LIN {X 0,Y 536.387,Z 823.114,A -85,B 0,C 180,E1 -258.059,E2 -258.059} C_VEL
LIN {X 0,Y 536.157,Z 833.006,A -85,B 0,C 180,E1 -259.949,E2 -259.949} C_VEL
LIN {X 0,Y 536.017,Z 840.915,A -85,B 0,C 180,E1 -261.85,E2 -261.85} C_VEL
LIN {X 0,Y 535.953,Z 847.088,A -85,B 0,C 180,E1 -263.789,E2 -263.789} C_VEL
LIN {X 0,Y 535.924,Z 851.492,A -85,B 0,C 180,E1 -265.721,E2 -265.721} C_VEL
LIN {X 0,Y 535.914,Z 854.356,A -85,B 0,C 180,E1 -267.755,E2 -267.755} C_VEL
LIN {X 0,Y 535.911,Z 855.453,A -85,B 0,C 180,E1 -269.787,E2 -269.787} C_VEL
LIN {X 0,Y 535.913,Z 854.809,A -85,B 0,C 180,E1 -271.818,E2 -271.818} C_VEL
LIN {X 0,Y 535.915,Z 852.571,A -85,B 0,C 180,E1 -273.744,E2 -273.744} C_VEL
LIN {X 0,Y 535.934,Z 848.705,A -85,B 0,C 180,E1 -275.675,E2 -275.675} C_VEL
LIN {X 0,Y 535.992,Z 843.122,A -85,B 0,C 180,E1 -277.611,E2 -277.611} C_VEL
LIN {X 0,Y 536.104,Z 835.67,A -85,B 0,C 180,E1 -279.555,E2 -279.555} C_VEL
LIN {X 0,Y 536.296,Z 826.694,A -85,B 0,C 180,E1 -281.398,E2 -281.398} C_VEL
LIN {X 0,Y 536.575,Z 816.255,A -85,B 0,C 180,E1 -283.141,E2 -283.141} C_VEL
LIN {X 0,Y 536.94,Z 804.373,A -85,B 0,C 180,E1 -284.781,E2 -284.781} C_VEL
LIN {X 0,Y 537.402,Z 790.987,A -85,B 0,C 180,E1 -286.317,E2 -286.317} C_VEL
LIN {X 0,Y 537.942,Z 775.934,A -85,B 0,C 180,E1 -287.748,E2 -287.748} C_VEL
LIN {X 0,Y 538.493,Z 760.519,A -85,B 0,C 180,E1 -288.962,E2 -288.962} C_VEL
LIN {X 0,Y 539.019,Z 744.186,A -85,B 0,C 180,E1 -290.019,E2 -290.019} C_VEL
LIN {X 0,Y 539.579,Z 727.091,A -85,B 0,C 180,E1 -290.904,E2 -290.904} C_VEL
LIN {X 0,Y 540.061,Z 708.873,A -85,B 0,C 180,E1 -291.632,E2 -291.632} C_VEL
LIN {X 0,Y 540.458,Z 689.501,A -85,B 0,C 180,E1 -292.184,E2 -292.184} C_VEL
LIN {X 0,Y 540.712,Z 668.628,A -85,B 0,C 180,E1 -292.553,E2 -292.553} C_VEL
LIN {X 0,Y 541.759,Z 481.528,A -85,B 0,C 180,E1 -295.18,E2 -295.18} C_VEL
LIN {X 0,Y 540.704,Z 474.497,A -85,B 0,C 180,E1 -295.347,E2 -295.347} C_VEL
LIN {X 0,Y 541.808,Z 432.243,A -85,B 0,C 180,E1 -298.432,E2 -298.432} C_VEL
LIN {X 0,Y 542.888,Z 388.213,A -85,B 0,C 180,E1 -301.662,E2 -301.662} C_VEL
LIN {X 0,Y 542.864,Z 381.603,A -85,B 0,C 180,E1 -302.16,E2 -302.16} C_VEL
LIN {X 0,Y 536.405,Z 363.919,A -85,B 0,C 180,E1 -303.915,E2 -303.915} C_VEL
LIN {X 0,Y 536.456,Z 363.914,A -85,B 0,C 180,E1 -307.264,E2 -307.264} C_VEL
LIN {X 0,Y 536.412,Z 363.912,A -85,B 0,C 180,E1 -310.491,E2 -310.491} C_VEL
LIN {X 0,Y 536.412,Z 363.907,A -85,B 0,C 180,E1 -313.987,E2 -313.987} C_VEL
LIN {X 0,Y 536.457,Z 363.908,A -85,B 0,C 180,E1 -317.252,E2 -317.252} C_VEL
LIN {X 0,Y 536.403,Z 363.915,A -85,B 0,C 180,E1 -320.533,E2 -320.533} C_VEL
LIN {X 0,Y 536.486,Z 364.089,A -85,B 0,C 180,E1 -323.676,E2 -323.676} C_VEL
LIN {X 0,Y 544.504,Z 385.078,A -85,B 0,C 180,E1 -326.099,E2 -326.099} C_VEL
LIN {X 0,Y 543.343,Z 422.568,A -85,B 0,C 180,E1 -329.108,E2 -329.108} C_VEL
LIN {X 0,Y 541.867,Z 466.231,A -85,B 0,C 180,E1 -332.567,E2 -332.567} C_VEL
LIN {X 0,Y 540.509,Z 512.697,A -85,B 0,C 180,E1 -336.159,E2 -336.159} C_VEL
LIN {X 0,Y 539.079,Z 559.766,A -85,B 0,C 180,E1 -339.803,E2 -339.803} C_VEL
LIN {X 0,Y 538.459,Z 589.965,A -85,B 0,C 180,E1 -342.057,E2 -342.057} C_VEL
LIN {X 0,Y 539.022,Z 598.616,A -85,B 0,C 180,E1 -342.216,E2 -342.216} C_VEL
LIN {X 0,Y 538.33,Z 729.225,A -85,B 0,C 180,E1 -344.027,E2 -344.027} C_VEL
LIN {X 0,Y 538.167,Z 742.956,A -85,B 0,C 180,E1 -344.34,E2 -344.34} C_VEL
LIN {X 0,Y 537.937,Z 758.206,A -85,B 0,C 180,E1 -344.862,E2 -344.862} C_VEL
LIN {X 0,Y 537.587,Z 772.683,A -85,B 0,C 180,E1 -345.568,E2 -345.568} C_VEL
LIN {X 0,Y 537.284,Z 784.959,A -85,B 0,C 180,E1 -346.329,E2 -346.329} C_VEL
LIN {X 0,Y 536.974,Z 797.896,A -85,B 0,C 180,E1 -347.307,E2 -347.307} C_VEL
LIN {X 0,Y 536.642,Z 810.315,A -85,B 0,C 180,E1 -348.5,E2 -348.5} C_VEL
LIN {X 0,Y 536.416,Z 819.61,A -85,B 0,C 180,E1 -349.583,E2 -349.583} C_VEL
LIN {X 0,Y 536.231,Z 828.137,A -85,B 0,C 180,E1 -350.772,E2 -350.772} C_VEL
LIN {X 0,Y 536.079,Z 836.92,A -85,B 0,C 180,E1 -352.282,E2 -352.282} C_VEL
LIN {X 0,Y 535.984,Z 843.614,A -85,B 0,C 180,E1 -353.788,E2 -353.788} C_VEL
LIN {X 0,Y 535.941,Z 848.401,A -85,B 0,C 180,E1 -355.184,E2 -355.184} C_VEL
LIN {X 0,Y 535.919,Z 852.383,A -85,B 0,C 180,E1 -356.791,E2 -356.791} C_VEL
LIN {X 0,Y 535.916,Z 854.749,A -85,B 0,C 180,E1 -358.503,E2 -358.503} C_VEL
LIN {X 0,Y 535.917,Z 855.42,A -85,B 0,C 180,E1 -360,E2 -360} C_VEL
LIN {X 0,Y 535.915,Z 854.816,A -85,B 0,C 180,E1 -361.496,E2 -361.496} C_VEL
LIN {X 0,Y 535.921,Z 852.56,A -85,B 0,C 180,E1 -363.208,E2 -363.208} C_VEL
LIN {X 0,Y 535.941,Z 848.675,A -85,B 0,C 180,E1 -364.815,E2 -364.815} C_VEL
LIN {X 0,Y 535.978,Z 843.962,A -85,B 0,C 180,E1 -366.211,E2 -366.211} C_VEL
LIN {X 0,Y 536.062,Z 837.86,A -85,B 0,C 180,E1 -367.61,E2 -367.61} C_VEL
LIN {X 0,Y 536.223,Z 828.743,A -85,B 0,C 180,E1 -369.227,E2 -369.227} C_VEL
LIN {X 0,Y 536.4,Z 820.32,A -85,B 0,C 180,E1 -370.417,E2 -370.417} C_VEL
LIN {X 0,Y 536.62,Z 811.143,A -85,B 0,C 180,E1 -371.5,E2 -371.5} C_VEL
LIN {X 0,Y 536.925,Z 799.619,A -85,B 0,C 180,E1 -372.631,E2 -372.631} C_VEL
LIN {X 0,Y 537.274,Z 785.525,A -85,B 0,C 180,E1 -373.726,E2 -373.726} C_VEL
LIN {X 0,Y 537.565,Z 774.465,A -85,B 0,C 180,E1 -374.432,E2 -374.432} C_VEL
LIN {X 0,Y 537.878,Z 761.699,A -85,B 0,C 180,E1 -375.084,E2 -375.084} C_VEL
LIN {X 0,Y 538.172,Z 745.734,A -85,B 0,C 180,E1 -375.687,E2 -375.687} C_VEL
LIN {X 0,Y 538.345,Z 730.703,A -85,B 0,C 180,E1 -376.048,E2 -376.048} C_VEL
LIN {X 0,Y 539.112,Z 638.988,A -85,B 0,C 180,E1 -377.399,E2 -377.399} C_VEL
LIN {X 0,Y 539.332,Z 593.98,A -85,B 0,C 180,E1 -378.066,E2 -378.066} C_VEL
LIN {X 0,Y 539.288,Z 591.918,A -85,B 0,C 180,E1 -378.148,E2 -378.148} C_VEL
LIN {X 0,Y 541.136,Z 554.692,A -85,B 0,C 180,E1 -381.175,E2 -381.175} C_VEL
LIN {X 0,Y 544.018,Z 511.719,A -85,B 0,C 180,E1 -384.778,E2 -384.778} C_VEL
LIN {X 0,Y 547.31,Z 475.035,A -85,B 0,C 180,E1 -388.002,E2 -388.002} C_VEL
LIN {X 0,Y 551.674,Z 441.606,A -85,B 0,C 180,E1 -391.1,E2 -391.1} C_VEL
LIN {X 0,Y 556.543,Z 416.023,A -85,B 0,C 180,E1 -393.658,E2 -393.658} C_VEL
LIN {X 0,Y 558.549,Z 407.726,A -85,B 0,C 180,E1 -394.573,E2 -394.573} C_VEL
LIN {X 0,Y 559.455,Z 403.927,A -85,B 0,C 180,E1 -395.061,E2 -395.061} C_VEL
LIN {X 0,Y 558.872,Z 401.471,A -85,B 0,C 180,E1 -395.931,E2 -395.931} C_VEL
LIN {X 0,Y 558.829,Z 399.609,A -85,B 0,C 180,E1 -397.082,E2 -397.082} C_VEL
LIN {X 0,Y 559.096,Z 399.371,A -85,B 0,C 180,E1 -397.474,E2 -397.474} C_VEL
LIN {X 0,Y 554.148,Z 410.442,A -85,B 0,C 180,E1 -398.498,E2 -398.498} C_VEL
LIN {X 0,Y 550.307,Z 424.122,A -85,B 0,C 180,E1 -399.623,E2 -399.623} C_VEL
LIN {X 0,Y 547.791,Z 440.126,A -85,B 0,C 180,E1 -400.829,E2 -400.829} C_VEL
LIN {X 0,Y 547.322,Z 456.11,A -85,B 0,C 180,E1 -402.023,E2 -402.023} C_VEL
LIN {X 0,Y 548.928,Z 469.64,A -85,B 0,C 180,E1 -403.082,E2 -403.082} C_VEL
LIN {X 0,Y 552.062,Z 480.529,A -85,B 0,C 180,E1 -403.993,E2 -403.993} C_VEL
LIN {X 0,Y 556.38,Z 489.245,A -85,B 0,C 180,E1 -404.785,E2 -404.785} C_VEL
LIN {X 0,Y 562.574,Z 497.444,A -85,B 0,C 180,E1 -405.6,E2 -405.6} C_VEL
LIN {X 0,Y 569.615,Z 503.816,A -85,B 0,C 180,E1 -406.318,E2 -406.318} C_VEL
LIN {X 0,Y 577.113,Z 508.538,A -85,B 0,C 180,E1 -406.98,E2 -406.98} C_VEL
LIN {X 0,Y 581.203,Z 510.142,A -85,B 0,C 180,E1 -407.461,E2 -407.461} C_VEL
LIN {X 0,Y 584.395,Z 510.594,A -85,B 0,C 180,E1 -408.012,E2 -408.012} C_VEL
LIN {X 0,Y 586.46,Z 509.917,A -85,B 0,C 180,E1 -408.604,E2 -408.604} C_VEL
LIN {X 0,Y 587.224,Z 508.161,A -85,B 0,C 180,E1 -409.215,E2 -409.215} C_VEL
LIN {X 0,Y 586.511,Z 505.309,A -85,B 0,C 180,E1 -409.815,E2 -409.815} C_VEL
LIN {X 0,Y 584.311,Z 501.673,A -85,B 0,C 180,E1 -410.337,E2 -410.337} C_VEL
LIN {X 0,Y 578.602,Z 493.885,A -85,B 0,C 180,E1 -411.054,E2 -411.054} C_VEL
LIN {X 0,Y 573.375,Z 484.319,A -85,B 0,C 180,E1 -411.705,E2 -411.705} C_VEL
LIN {X 0,Y 569.141,Z 473.459,A -85,B 0,C 180,E1 -412.248,E2 -412.248} C_VEL
LIN {X 0,Y 565.904,Z 461.458,A -85,B 0,C 180,E1 -412.673,E2 -412.673} C_VEL
LIN {X 0,Y 564.883,Z 456.447,A -85,B 0,C 180,E1 -412.809,E2 -412.809} C_VEL
LIN {X 0,Y 562.174,Z 463.362,A -85,B 0,C 180,E1 -413.175,E2 -413.175} C_VEL
LIN {X 0,Y 559.86,Z 469.22,A -85,B 0,C 180,E1 -413.492,E2 -413.492} C_VEL
LIN {X 0,Y 558.97,Z 470.969,A -85,B 0,C 180,E1 -413.615,E2 -413.615} C_VEL
LIN {X 0,Y 554.81,Z 519.429,A -85,B 0,C 180,E1 -414.203,E2 -414.203} C_VEL
LIN {X 0,Y 551.082,Z 552.372,A -85,B 0,C 180,E1 -414.744,E2 -414.744} C_VEL
LIN {X 0,Y 548.664,Z 567.257,A -85,B 0,C 180,E1 -415.102,E2 -415.102} C_VEL
LIN {X 0,Y 547.486,Z 570.982,A -85,B 0,C 180,E1 -415.279,E2 -415.279} C_VEL
LIN {X 0,Y 547.134,Z 571.563,A -85,B 0,C 180,E1 -415.337,E2 -415.337} C_VEL
LIN {X 0,Y 545.349,Z 761.519,A -85,B 0,C 180,E1 -418.174,E2 -418.174} C_VEL
LIN {X 0,Y 544.771,Z 783.502,A -85,B 0,C 180,E1 -418.695,E2 -418.695} C_VEL
LIN {X 0,Y 544.053,Z 806.31,A -85,B 0,C 180,E1 -419.459,E2 -419.459} C_VEL
LIN {X 0,Y 543.205,Z 827.548,A -85,B 0,C 180,E1 -420.381,E2 -420.381} C_VEL
LIN {X 0,Y 542.286,Z 847.779,A -85,B 0,C 180,E1 -421.475,E2 -421.475} C_VEL
LIN {X 0,Y 541.287,Z 867.98,A -85,B 0,C 180,E1 -422.794,E2 -422.794} C_VEL
LIN {X 0,Y 540.249,Z 887.816,A -85,B 0,C 180,E1 -424.337,E2 -424.337} C_VEL
LIN {X 0,Y 539.331,Z 905.831,A -85,B 0,C 180,E1 -425.988,E2 -425.988} C_VEL
LIN {X 0,Y 538.461,Z 923.22,A -85,B 0,C 180,E1 -427.855,E2 -427.855} C_VEL
LIN {X 0,Y 537.693,Z 939.401,A -85,B 0,C 180,E1 -429.894,E2 -429.894} C_VEL
LIN {X 0,Y 537.082,Z 953.596,A -85,B 0,C 180,E1 -431.999,E2 -431.999} C_VEL
LIN {X 0,Y 536.623,Z 966.268,A -85,B 0,C 180,E1 -434.214,E2 -434.214} C_VEL
LIN {X 0,Y 536.313,Z 976.854,A -85,B 0,C 180,E1 -436.414,E2 -436.414} C_VEL
LIN {X 0,Y 536.107,Z 985.923,A -85,B 0,C 180,E1 -438.707,E2 -438.707} C_VEL
LIN {X 0,Y 535.994,Z 993.093,A -85,B 0,C 180,E1 -440.985,E2 -440.985} C_VEL
LIN {X 0,Y 535.942,Z 998.591,A -85,B 0,C 180,E1 -443.25,E2 -443.25} C_VEL
LIN {X 0,Y 535.921,Z 1002.584,A -85,B 0,C 180,E1 -445.613,E2 -445.613} C_VEL
LIN {X 0,Y 535.911,Z 1004.832,A -85,B 0,C 180,E1 -447.968,E2 -447.968} C_VEL
LIN {X 0,Y 535.894,Z 1005.442,A -85,B 0,C 180,E1 -450.427,E2 -450.427} C_VEL
LIN {X 0,Y 535.894,Z 1004.424,A -85,B 0,C 180,E1 -452.673,E2 -452.673} C_VEL
LIN {X 0,Y 535.901,Z 1001.8,A -85,B 0,C 180,E1 -454.926,E2 -454.926} C_VEL
LIN {X 0,Y 535.929,Z 997.683,A -85,B 0,C 180,E1 -457.18,E2 -457.18} C_VEL
LIN {X 0,Y 535.997,Z 991.879,A -85,B 0,C 180,E1 -459.448,E2 -459.448} C_VEL
LIN {X 0,Y 536.128,Z 984.297,A -85,B 0,C 180,E1 -461.735,E2 -461.735} C_VEL
LIN {X 0,Y 536.357,Z 974.911,A -85,B 0,C 180,E1 -464.025,E2 -464.025} C_VEL
LIN {X 0,Y 536.693,Z 963.937,A -85,B 0,C 180,E1 -466.227,E2 -466.227} C_VEL
LIN {X 0,Y 537.16,Z 951.48,A -85,B 0,C 180,E1 -468.335,E2 -468.335} C_VEL
LIN {X 0,Y 537.766,Z 937.595,A -85,B 0,C 180,E1 -470.346,E2 -470.346} C_VEL
LIN {X 0,Y 538.505,Z 922.234,A -85,B 0,C 180,E1 -472.257,E2 -472.257} C_VEL
LIN {X 0,Y 539.363,Z 905.276,A -85,B 0,C 180,E1 -474.068,E2 -474.068} C_VEL
LIN {X 0,Y 540.321,Z 886.47,A -85,B 0,C 180,E1 -475.776,E2 -475.776} C_VEL
LIN {X 0,Y 541.326,Z 867.187,A -85,B 0,C 180,E1 -477.262,E2 -477.262} C_VEL
LIN {X 0,Y 542.328,Z 846.795,A -85,B 0,C 180,E1 -478.582,E2 -478.582} C_VEL
LIN {X 0,Y 543.204,Z 827.56,A -85,B 0,C 180,E1 -479.618,E2 -479.618} C_VEL
LIN {X 0,Y 544.053,Z 806.327,A -85,B 0,C 180,E1 -480.54,E2 -480.54} C_VEL
LIN {X 0,Y 544.782,Z 783.156,A -85,B 0,C 180,E1 -481.315,E2 -481.315} C_VEL
LIN {X 0,Y 545.362,Z 761.024,A -85,B 0,C 180,E1 -481.836,E2 -481.836} C_VEL
LIN {X 0,Y 547.27,Z 571.184,A -85,B 0,C 180,E1 -484.688,E2 -484.688} C_VEL
LIN {X 0,Y 548.267,Z 568.899,A -85,B 0,C 180,E1 -484.838,E2 -484.838} C_VEL
LIN {X 0,Y 550.436,Z 557.003,A -85,B 0,C 180,E1 -485.161,E2 -485.161} C_VEL
LIN {X 0,Y 553.985,Z 527.566,A -85,B 0,C 180,E1 -485.679,E2 -485.679} C_VEL
LIN {X 0,Y 558.161,Z 481.457,A -85,B 0,C 180,E1 -486.272,E2 -486.272} C_VEL
LIN {X 0,Y 559.115,Z 470.446,A -85,B 0,C 180,E1 -486.405,E2 -486.405} C_VEL
LIN {X 0,Y 561.46,Z 465.551,A -85,B 0,C 180,E1 -486.728,E2 -486.728} C_VEL
LIN {X 0,Y 563.371,Z 460.11,A -85,B 0,C 180,E1 -486.988,E2 -486.988} C_VEL
LIN {X 0,Y 564.936,Z 456.583,A -85,B 0,C 180,E1 -487.198,E2 -487.198} C_VEL
LIN {X 0,Y 567.839,Z 469.202,A -85,B 0,C 180,E1 -487.582,E2 -487.582} C_VEL
LIN {X 0,Y 571.748,Z 480.579,A -85,B 0,C 180,E1 -488.088,E2 -488.088} C_VEL
LIN {X 0,Y 576.639,Z 490.657,A -85,B 0,C 180,E1 -488.704,E2 -488.704} C_VEL
LIN {X 0,Y 582.546,Z 499.398,A -85,B 0,C 180,E1 -489.424,E2 -489.424} C_VEL
LIN {X 0,Y 585.465,Z 503.391,A -85,B 0,C 180,E1 -489.884,E2 -489.884} C_VEL
LIN {X 0,Y 586.997,Z 506.612,A -85,B 0,C 180,E1 -490.429,E2 -490.429} C_VEL
LIN {X 0,Y 587.094,Z 508.969,A -85,B 0,C 180,E1 -491.022,E2 -491.022} C_VEL
LIN {X 0,Y 585.831,Z 510.295,A -85,B 0,C 180,E1 -491.622,E2 -491.622} C_VEL
LIN {X 0,Y 583.164,Z 510.544,A -85,B 0,C 180,E1 -492.229,E2 -492.229} C_VEL
LIN {X 0,Y 579.798,Z 509.694,A -85,B 0,C 180,E1 -492.724,E2 -492.724} C_VEL
LIN {X 0,Y 571.887,Z 505.541,A -85,B 0,C 180,E1 -493.63,E2 -493.63} C_VEL
LIN {X 0,Y 565.274,Z 499.908,A -85,B 0,C 180,E1 -494.535,E2 -494.535} C_VEL
LIN {X 0,Y 560.009,Z 492.953,A -85,B 0,C 180,E1 -495.439,E2 -495.439} C_VEL
LIN {X 0,Y 555.868,Z 484.228,A -85,B 0,C 180,E1 -496.385,E2 -496.385} C_VEL
LIN {X 0,Y 553.159,Z 473.762,A -85,B 0,C 180,E1 -497.363,E2 -497.363} C_VEL
LIN {X 0,Y 551.719,Z 460.276,A -85,B 0,C 180,E1 -498.457,E2 -498.457} C_VEL
LIN {X 0,Y 551.957,Z 441.599,A -85,B 0,C 180,E1 -499.775,E2 -499.775} C_VEL
LIN {X 0,Y 553.891,Z 401.672,A -85,B 0,C 180,E1 -502.531,E2 -502.531} C_VEL
LIN {X 0,Y 554.042,Z 396.212,A -85,B 0,C 180,E1 -502.933,E2 -502.933} C_VEL
LIN {X 0,Y 546.158,Z 382.054,A -85,B 0,C 180,E1 -505.04,E2 -505.04} C_VEL
LIN {X 0,Y 541.163,Z 373.11,A -85,B 0,C 180,E1 -506.436,E2 -506.436} C_VEL
LIN {X 0,Y 539.331,Z 369.712,A -85,B 0,C 180,E1 -506.973,E2 -506.973} C_VEL
LIN {X 0,Y 536.8,Z 365.411,A -85,B 0,C 180,E1 -507.685,E2 -507.685} C_VEL
LIN {X 0,Y 536.468,Z 363.913,A -85,B 0,C 180,E1 -507.87,E2 -507.87} C_VEL
LIN {X 0,Y 536.425,Z 363.915,A -85,B 0,C 180,E1 -511.257,E2 -511.257} C_VEL
LIN {X 0,Y 536.433,Z 363.914,A -85,B 0,C 180,E1 -514.852,E2 -514.852} C_VEL
LIN {X 0,Y 536.465,Z 363.91,A -85,B 0,C 180,E1 -518.23,E2 -518.23} C_VEL
LIN {X 0,Y 536.442,Z 363.914,A -85,B 0,C 180,E1 -521.752,E2 -521.752} C_VEL
LIN {X 0,Y 536.466,Z 363.912,A -85,B 0,C 180,E1 -525.096,E2 -525.096} C_VEL
LIN {X 0,Y 536.46,Z 363.913,A -85,B 0,C 180,E1 -528.497,E2 -528.497} C_VEL
LIN {X 0,Y 536.458,Z 363.913,A -85,B 0,C 180,E1 -531.857,E2 -531.857} C_VEL
LIN {X 0,Y 536.44,Z 363.917,A -85,B 0,C 180,E1 -535.189,E2 -535.189} C_VEL
LIN {X 0,Y 536.461,Z 363.914,A -85,B 0,C 180,E1 -538.505,E2 -538.505} C_VEL
LIN {X 0,Y 536.422,Z 363.918,A -85,B 0,C 180,E1 -541.923,E2 -541.923} C_VEL
LIN {X 0,Y 536.455,Z 363.911,A -85,B 0,C 180,E1 -545.348,E2 -545.348} C_VEL
LIN {X 0,Y 536.43,Z 363.915,A -85,B 0,C 180,E1 -548.684,E2 -548.684} C_VEL
LIN {X 0,Y 536.427,Z 363.915,A -85,B 0,C 180,E1 -552.159,E2 -552.159} C_VEL
LIN {X 0,Y 536.466,Z 363.909,A -85,B 0,C 180,E1 -555.569,E2 -555.569} C_VEL
LIN {X 0,Y 536.438,Z 363.914,A -85,B 0,C 180,E1 -559.037,E2 -559.037} C_VEL
LIN {X 0,Y 536.465,Z 363.914,A -85,B 0,C 180,E1 -562.463,E2 -562.463} C_VEL
LIN {X 0,Y 536.459,Z 363.913,A -85,B 0,C 180,E1 -565.858,E2 -565.858} C_VEL
LIN {X 0,Y 536.457,Z 363.913,A -85,B 0,C 180,E1 -569.277,E2 -569.277} C_VEL
LIN {X 0,Y 536.432,Z 363.916,A -85,B 0,C 180,E1 -572.597,E2 -572.597} C_VEL
LIN {X 0,Y 536.433,Z 363.91,A -85,B 0,C 180,E1 -574.588,E2 -574.588} C_VEL
LIN {X 0,Y 535.428,Z 364.033,A -85,B 0,C 180,E1 -575.411,E2 -575.411} C_VEL
LIN {X 0,Y 529.04,Z 364.829,A -85,B 0,C 180,E1 -577.723,E2 -577.723} C_VEL
LIN {X 0,Y 528.526,Z 364.894,A -85,B 0,C 180,E1 -578.325,E2 -578.325} C_VEL
LIN {X 0,Y 528.504,Z 364.893,A -85,B 0,C 180,E1 -581.807,E2 -581.807} C_VEL
LIN {X 0,Y 528.523,Z 364.905,A -85,B 0,C 180,E1 -585.188,E2 -585.188} C_VEL
LIN {X 0,Y 528.521,Z 364.904,A -85,B 0,C 180,E1 -588.682,E2 -588.682} C_VEL
LIN {X 0,Y 528.513,Z 364.899,A -85,B 0,C 180,E1 -592.083,E2 -592.083} C_VEL
LIN {X 0,Y 528.479,Z 364.909,A -85,B 0,C 180,E1 -595.55,E2 -595.55} C_VEL
LIN {X 0,Y 528.496,Z 365.068,A -85,B 0,C 180,E1 -595.715,E2 -595.715} C_VEL
LIN {X 0,Y 535.912,Z 384.982,A -85,B 0,C 180,E1 -597.708,E2 -597.708} C_VEL
LIN {X 0,Y 534.68,Z 430.458,A -85,B 0,C 180,E1 -601.087,E2 -601.087} C_VEL
LIN {X 0,Y 533.602,Z 476.361,A -85,B 0,C 180,E1 -604.403,E2 -604.403} C_VEL
LIN {X 0,Y 534.725,Z 485.378,A -85,B 0,C 180,E1 -604.596,E2 -604.596} C_VEL
LIN {X 0,Y 533.229,Z 683.64,A -85,B 0,C 180,E1 -607.434,E2 -607.434} C_VEL
LIN {X 0,Y 532.889,Z 701.992,A -85,B 0,C 180,E1 -607.885,E2 -607.885} C_VEL
LIN {X 0,Y 532.411,Z 719.706,A -85,B 0,C 180,E1 -608.518,E2 -608.518} C_VEL
LIN {X 0,Y 531.792,Z 737.309,A -85,B 0,C 180,E1 -609.358,E2 -609.358} C_VEL
LIN {X 0,Y 531.116,Z 753.841,A -85,B 0,C 180,E1 -610.365,E2 -610.365} C_VEL
LIN {X 0,Y 530.393,Z 771.626,A -85,B 0,C 180,E1 -611.707,E2 -611.707} C_VEL
LIN {X 0,Y 529.791,Z 786.298,A -85,B 0,C 180,E1 -613.048,E2 -613.048} C_VEL
LIN {X 0,Y 529.247,Z 800.016,A -85,B 0,C 180,E1 -614.551,E2 -614.551} C_VEL
LIN {X 0,Y 528.786,Z 812.65,A -85,B 0,C 180,E1 -616.217,E2 -616.217} C_VEL
LIN {X 0,Y 528.433,Z 823.943,A -85,B 0,C 180,E1 -618.023,E2 -618.023} C_VEL
LIN {X 0,Y 528.187,Z 833.309,A -85,B 0,C 180,E1 -619.861,E2 -619.861} C_VEL
LIN {X 0,Y 528.038,Z 840.916,A -85,B 0,C 180,E1 -621.726,E2 -621.726} C_VEL
LIN {X 0,Y 527.958,Z 847.09,A -85,B 0,C 180,E1 -623.694,E2 -623.694} C_VEL
LIN {X 0,Y 527.925,Z 851.494,A -85,B 0,C 180,E1 -625.656,E2 -625.656} C_VEL
LIN {X 0,Y 527.913,Z 854.356,A -85,B 0,C 180,E1 -627.721,E2 -627.721} C_VEL
LIN {X 0,Y 527.911,Z 855.453,A -85,B 0,C 180,E1 -629.783,E2 -629.783} C_VEL
LIN {X 0,Y 527.913,Z 854.808,A -85,B 0,C 180,E1 -631.845,E2 -631.845} C_VEL
LIN {X 0,Y 527.918,Z 852.57,A -85,B 0,C 180,E1 -633.801,E2 -633.801} C_VEL
LIN {X 0,Y 527.937,Z 848.704,A -85,B 0,C 180,E1 -635.761,E2 -635.761} C_VEL
LIN {X 0,Y 528.007,Z 843.119,A -85,B 0,C 180,E1 -637.727,E2 -637.727} C_VEL
LIN {X 0,Y 528.134,Z 835.669,A -85,B 0,C 180,E1 -639.701,E2 -639.701} C_VEL
LIN {X 0,Y 528.354,Z 826.693,A -85,B 0,C 180,E1 -641.572,E2 -641.572} C_VEL
LIN {X 0,Y 528.674,Z 816.253,A -85,B 0,C 180,E1 -643.341,E2 -643.341} C_VEL
LIN {X 0,Y 529.111,Z 803.908,A -85,B 0,C 180,E1 -645.063,E2 -645.063} C_VEL
LIN {X 0,Y 529.633,Z 790.432,A -85,B 0,C 180,E1 -646.619,E2 -646.619} C_VEL
LIN {X 0,Y 530.222,Z 775.924,A -85,B 0,C 180,E1 -648.015,E2 -648.015} C_VEL
LIN {X 0,Y 530.88,Z 759.69,A -85,B 0,C 180,E1 -649.307,E2 -649.307} C_VEL
LIN {X 0,Y 531.528,Z 743.735,A -85,B 0,C 180,E1 -650.366,E2 -650.366} C_VEL
LIN {X 0,Y 532.184,Z 726.55,A -85,B 0,C 180,E1 -651.27,E2 -651.27} C_VEL
LIN {X 0,Y 532.732,Z 708.036,A -85,B 0,C 180,E1 -652.011,E2 -652.011} C_VEL
LIN {X 0,Y 533.133,Z 689.61,A -85,B 0,C 180,E1 -652.531,E2 -652.531} C_VEL
LIN {X 0,Y 533.377,Z 668.55,A -85,B 0,C 180,E1 -652.897,E2 -652.897} C_VEL
LIN {X 0,Y 534.562,Z 482.581,A -85,B 0,C 180,E1 -655.544,E2 -655.544} C_VEL
LIN {X 0,Y 533.518,Z 475.565,A -85,B 0,C 180,E1 -655.719,E2 -655.719} C_VEL
LIN {X 0,Y 534.694,Z 430.123,A -85,B 0,C 180,E1 -659.03,E2 -659.03} C_VEL
LIN {X 0,Y 535.897,Z 385.079,A -85,B 0,C 180,E1 -662.377,E2 -662.377} C_VEL
LIN {X 0,Y 529.73,Z 368.431,A -85,B 0,C 180,E1 -664.044,E2 -664.044} C_VEL
LIN {X 0,Y 528.481,Z 364.904,A -85,B 0,C 180,E1 -664.405,E2 -664.405} C_VEL
LIN {X 0,Y 528.473,Z 364.904,A -85,B 0,C 180,E1 -667.807,E2 -667.807} C_VEL
LIN {X 0,Y 528.521,Z 364.895,A -85,B 0,C 180,E1 -671.031,E2 -671.031} C_VEL
LIN {X 0,Y 528.466,Z 364.896,A -85,B 0,C 180,E1 -674.342,E2 -674.342} C_VEL
LIN {X 0,Y 528.509,Z 364.892,A -85,B 0,C 180,E1 -677.707,E2 -677.707} C_VEL
LIN {X 0,Y 528.479,Z 364.898,A -85,B 0,C 180,E1 -680.948,E2 -680.948} C_VEL
LIN {X 0,Y 528.518,Z 365.148,A -85,B 0,C 180,E1 -683.093,E2 -683.093} C_VEL
LIN {X 0,Y 537.22,Z 387.368,A -85,B 0,C 180,E1 -685.727,E2 -685.727} C_VEL
LIN {X 0,Y 537.491,Z 389.74,A -85,B 0,C 180,E1 -685.949,E2 -685.949} C_VEL
LIN {X 0,Y 536.131,Z 429.265,A -85,B 0,C 180,E1 -689.145,E2 -689.145} C_VEL
LIN {X 0,Y 534.525,Z 472.595,A -85,B 0,C 180,E1 -692.602,E2 -692.602} C_VEL
LIN {X 0,Y 533.057,Z 517.272,A -85,B 0,C 180,E1 -696.099,E2 -696.099} C_VEL
LIN {X 0,Y 531.6,Z 563.498,A -85,B 0,C 180,E1 -699.695,E2 -699.695} C_VEL
LIN {X 0,Y 530.993,Z 590.742,A -85,B 0,C 180,E1 -701.746,E2 -701.746} C_VEL
LIN {X 0,Y 531.581,Z 599.108,A -85,B 0,C 180,E1 -701.905,E2 -701.905} C_VEL
LIN {X 0,Y 530.718,Z 728.012,A -85,B 0,C 180,E1 -703.744,E2 -703.744} C_VEL
LIN {X 0,Y 530.542,Z 742.648,A -85,B 0,C 180,E1 -704.067,E2 -704.067} C_VEL
LIN {X 0,Y 530.302,Z 757.908,A -85,B 0,C 180,E1 -704.582,E2 -704.582} C_VEL
LIN {X 0,Y 529.94,Z 772.805,A -85,B 0,C 180,E1 -705.299,E2 -705.299} C_VEL
LIN {X 0,Y 529.602,Z 785.194,A -85,B 0,C 180,E1 -706.071,E2 -706.071} C_VEL
LIN {X 0,Y 529.238,Z 797.381,A -85,B 0,C 180,E1 -707.007,E2 -707.007} C_VEL
LIN {X 0,Y 528.844,Z 809.94,A -85,B 0,C 180,E1 -708.218,E2 -708.218} C_VEL
LIN {X 0,Y 528.525,Z 819.988,A -85,B 0,C 180,E1 -709.426,E2 -709.426} C_VEL
LIN {X 0,Y 528.291,Z 828.291,A -85,B 0,C 180,E1 -710.632,E2 -710.632} C_VEL
LIN {X 0,Y 528.092,Z 837.428,A -85,B 0,C 180,E1 -712.274,E2 -712.274} C_VEL
LIN {X 0,Y 527.994,Z 843.608,A -85,B 0,C 180,E1 -713.694,E2 -713.694} C_VEL
LIN {X 0,Y 527.946,Z 848.394,A -85,B 0,C 180,E1 -715.111,E2 -715.111} C_VEL
LIN {X 0,Y 527.92,Z 852.379,A -85,B 0,C 180,E1 -716.742,E2 -716.742} C_VEL
LIN {X 0,Y 527.915,Z 854.742,A -85,B 0,C 180,E1 -718.48,E2 -718.48} C_VEL
LIN {X 0,Y 527.917,Z 855.411,A -85,B 0,C 180,E1 -720,E2 -720} C_VEL
LIN {X 0,Y 527.915,Z 854.807,A -85,B 0,C 180,E1 -721.519,E2 -721.519} C_VEL
LIN {X 0,Y 527.922,Z 852.561,A -85,B 0,C 180,E1 -723.257,E2 -723.257} C_VEL
LIN {X 0,Y 527.944,Z 848.664,A -85,B 0,C 180,E1 -724.889,E2 -724.889} C_VEL
LIN {X 0,Y 527.988,Z 843.951,A -85,B 0,C 180,E1 -726.306,E2 -726.306} C_VEL
LIN {X 0,Y 528.084,Z 837.849,A -85,B 0,C 180,E1 -727.725,E2 -727.725} C_VEL
LIN {X 0,Y 528.293,Z 829.028,A -85,B 0,C 180,E1 -729.367,E2 -729.367} C_VEL
LIN {X 0,Y 528.535,Z 820.937,A -85,B 0,C 180,E1 -730.573,E2 -730.573} C_VEL
LIN {X 0,Y 528.83,Z 812.08,A -85,B 0,C 180,E1 -731.671,E2 -731.671} C_VEL
LIN {X 0,Y 529.23,Z 800.857,A -85,B 0,C 180,E1 -732.826,E2 -732.826} C_VEL
LIN {X 0,Y 529.666,Z 787.274,A -85,B 0,C 180,E1 -733.927,E2 -733.927} C_VEL
LIN {X 0,Y 530.03,Z 774.346,A -85,B 0,C 180,E1 -734.754,E2 -734.754} C_VEL
LIN {X 0,Y 530.393,Z 759.935,A -85,B 0,C 180,E1 -735.47,E2 -735.47} C_VEL
LIN {X 0,Y 530.63,Z 744.334,A -85,B 0,C 180,E1 -736.014,E2 -736.014} C_VEL
LIN {X 0,Y 530.795,Z 729.651,A -85,B 0,C 180,E1 -736.349,E2 -736.349} C_VEL
LIN {X 0,Y 531.93,Z 628.266,A -85,B 0,C 180,E1 -737.912,E2 -737.912} C_VEL
LIN {X 0,Y 532.287,Z 594.804,A -85,B 0,C 180,E1 -738.467,E2 -738.467} C_VEL
LIN {X 0,Y 534.096,Z 563.14,A -85,B 0,C 180,E1 -741.065,E2 -741.065} C_VEL
LIN {X 0,Y 536.74,Z 524.756,A -85,B 0,C 180,E1 -744.311,E2 -744.311} C_VEL
LIN {X 0,Y 540.608,Z 484.193,A -85,B 0,C 180,E1 -747.899,E2 -747.899} C_VEL
LIN {X 0,Y 544.696,Z 453.781,A -85,B 0,C 180,E1 -750.745,E2 -750.745} C_VEL
LIN {X 0,Y 549.942,Z 426.989,A -85,B 0,C 180,E1 -753.428,E2 -753.428} C_VEL
LIN {X 0,Y 553.677,Z 413.284,A -85,B 0,C 180,E1 -754.929,E2 -754.929} C_VEL
LIN {X 0,Y 554.683,Z 409.657,A -85,B 0,C 180,E1 -755.435,E2 -755.435} C_VEL
LIN {X 0,Y 554.418,Z 407.915,A -85,B 0,C 180,E1 -756.137,E2 -756.137} C_VEL
LIN {X 0,Y 554.593,Z 406.501,A -85,B 0,C 180,E1 -757.125,E2 -757.125} C_VEL
LIN {X 0,Y 548.964,Z 417.696,A -85,B 0,C 180,E1 -758.194,E2 -758.194} C_VEL
LIN {X 0,Y 544.511,Z 431.403,A -85,B 0,C 180,E1 -759.37,E2 -759.37} C_VEL
LIN {X 0,Y 541.796,Z 446.57,A -85,B 0,C 180,E1 -760.588,E2 -760.588} C_VEL
LIN {X 0,Y 541.209,Z 461.137,A -85,B 0,C 180,E1 -761.752,E2 -761.752} C_VEL
LIN {X 0,Y 542.67,Z 474.175,A -85,B 0,C 180,E1 -762.835,E2 -762.835} C_VEL
LIN {X 0,Y 545.848,Z 485.335,A -85,B 0,C 180,E1 -763.82,E2 -763.82} C_VEL
LIN {X 0,Y 550.314,Z 494.368,A -85,B 0,C 180,E1 -764.679,E2 -764.679} C_VEL
LIN {X 0,Y 556.383,Z 502.505,A -85,B 0,C 180,E1 -765.515,E2 -765.515} C_VEL
LIN {X 0,Y 564.055,Z 509.609,A -85,B 0,C 180,E1 -766.321,E2 -766.321} C_VEL
LIN {X 0,Y 573.177,Z 515.397,A -85,B 0,C 180,E1 -767.109,E2 -767.109} C_VEL
LIN {X 0,Y 577.397,Z 517.151,A -85,B 0,C 180,E1 -767.535,E2 -767.535} C_VEL
LIN {X 0,Y 580.887,Z 517.889,A -85,B 0,C 180,E1 -768.037,E2 -768.037} C_VEL
LIN {X 0,Y 583.542,Z 517.554,A -85,B 0,C 180,E1 -768.632,E2 -768.632} C_VEL
LIN {X 0,Y 584.877,Z 516.087,A -85,B 0,C 180,E1 -769.265,E2 -769.265} C_VEL
LIN {X 0,Y 584.68,Z 513.551,A -85,B 0,C 180,E1 -769.888,E2 -769.888} C_VEL
LIN {X 0,Y 582.927,Z 510.187,A -85,B 0,C 180,E1 -770.447,E2 -770.447} C_VEL
LIN {X 0,Y 579.389,Z 505.648,A -85,B 0,C 180,E1 -770.958,E2 -770.958} C_VEL
LIN {X 0,Y 573.143,Z 496.366,A -85,B 0,C 180,E1 -771.734,E2 -771.734} C_VEL
LIN {X 0,Y 568.071,Z 485.991,A -85,B 0,C 180,E1 -772.387,E2 -772.387} C_VEL
LIN {X 0,Y 563.939,Z 474.303,A -85,B 0,C 180,E1 -772.936,E2 -772.936} C_VEL
LIN {X 0,Y 563.751,Z 473.943,A -85,B 0,C 180,E1 -772.961,E2 -772.961} C_VEL
LIN {X 0,Y 563.347,Z 476.736,A -85,B 0,C 180,E1 -773.016,E2 -773.016} C_VEL
LIN {X 0,Y 559.081,Z 524.504,A -85,B 0,C 180,E1 -773.6,E2 -773.6} C_VEL
LIN {X 0,Y 555.341,Z 556.183,A -85,B 0,C 180,E1 -774.127,E2 -774.127} C_VEL
LIN {X 0,Y 552.879,Z 570.521,A -85,B 0,C 180,E1 -774.481,E2 -774.481} C_VEL
LIN {X 0,Y 551.421,Z 575.968,A -85,B 0,C 180,E1 -774.694,E2 -774.694} C_VEL
LIN {X 0,Y 547.205,Z 626.873,A -85,B 0,C 180,E1 -775.316,E2 -775.316} C_VEL
LIN {X 0,Y 544.154,Z 647.157,A -85,B 0,C 180,E1 -775.648,E2 -775.648} C_VEL
LIN {X 0,Y 541.182,Z 660.811,A -85,B 0,C 180,E1 -776.013,E2 -776.013} C_VEL
LIN {X 0,Y 539.577,Z 667.203,A -85,B 0,C 180,E1 -776.293,E2 -776.293} C_VEL
LIN {X 0,Y 538.542,Z 761.682,A -85,B 0,C 180,E1 -777.727,E2 -777.727} C_VEL
LIN {X 0,Y 537.908,Z 783.496,A -85,B 0,C 180,E1 -778.25,E2 -778.25} C_VEL
LIN {X 0,Y 537.108,Z 806.304,A -85,B 0,C 180,E1 -779.021,E2 -779.021} C_VEL
LIN {X 0,Y 536.16,Z 827.421,A -85,B 0,C 180,E1 -779.946,E2 -779.946} C_VEL
LIN {X 0,Y 535.133,Z 847.786,A -85,B 0,C 180,E1 -781.058,E2 -781.058} C_VEL
LIN {X 0,Y 534.006,Z 867.985,A -85,B 0,C 180,E1 -782.392,E2 -782.392} C_VEL
LIN {X 0,Y 532.849,Z 887.814,A -85,B 0,C 180,E1 -783.954,E2 -783.954} C_VEL
LIN {X 0,Y 531.812,Z 905.833,A -85,B 0,C 180,E1 -785.626,E2 -785.626} C_VEL
LIN {X 0,Y 530.82,Z 923.22,A -85,B 0,C 180,E1 -787.519,E2 -787.519} C_VEL
LIN {X 0,Y 529.956,Z 939.281,A -85,B 0,C 180,E1 -789.571,E2 -789.571} C_VEL
LIN {X 0,Y 529.254,Z 953.599,A -85,B 0,C 180,E1 -791.723,E2 -791.723} C_VEL
LIN {X 0,Y 528.723,Z 966.272,A -85,B 0,C 180,E1 -793.972,E2 -793.972} C_VEL
LIN {X 0,Y 528.37,Z 976.857,A -85,B 0,C 180,E1 -796.205,E2 -796.205} C_VEL
LIN {X 0,Y 528.136,Z 985.922,A -85,B 0,C 180,E1 -798.534,E2 -798.534} C_VEL
LIN {X 0,Y 528.006,Z 993.096,A -85,B 0,C 180,E1 -800.847,E2 -800.847} C_VEL
LIN {X 0,Y 527.942,Z 998.592,A -85,B 0,C 180,E1 -803.147,E2 -803.147} C_VEL
LIN {X 0,Y 527.919,Z 1002.585,A -85,B 0,C 180,E1 -805.546,E2 -805.546} C_VEL
LIN {X 0,Y 527.912,Z 1004.834,A -85,B 0,C 180,E1 -807.937,E2 -807.937} C_VEL
LIN {X 0,Y 527.894,Z 1005.445,A -85,B 0,C 180,E1 -810.434,E2 -810.434} C_VEL
LIN {X 0,Y 527.894,Z 1004.33,A -85,B 0,C 180,E1 -812.822,E2 -812.822} C_VEL
LIN {X 0,Y 527.9,Z 1001.648,A -85,B 0,C 180,E1 -815.107,E2 -815.107} C_VEL
LIN {X 0,Y 527.938,Z 997.194,A -85,B 0,C 180,E1 -817.509,E2 -817.509} C_VEL
LIN {X 0,Y 528.021,Z 991.252,A -85,B 0,C 180,E1 -819.812,E2 -819.812} C_VEL
LIN {X 0,Y 528.185,Z 983.509,A -85,B 0,C 180,E1 -822.129,E2 -822.129} C_VEL
LIN {X 0,Y 528.466,Z 973.876,A -85,B 0,C 180,E1 -824.462,E2 -824.462} C_VEL
LIN {X 0,Y 528.878,Z 962.746,A -85,B 0,C 180,E1 -826.7,E2 -826.7} C_VEL
LIN {X 0,Y 529.457,Z 949.347,A -85,B 0,C 180,E1 -828.954,E2 -828.954} C_VEL
LIN {X 0,Y 530.165,Z 934.977,A -85,B 0,C 180,E1 -831.007,E2 -831.007} C_VEL
LIN {X 0,Y 531.038,Z 918.949,A -85,B 0,C 180,E1 -832.971,E2 -832.971} C_VEL
LIN {X 0,Y 532.065,Z 901.316,A -85,B 0,C 180,E1 -834.818,E2 -834.818} C_VEL
LIN {X 0,Y 533.153,Z 883.048,A -85,B 0,C 180,E1 -836.449,E2 -836.449} C_VEL
LIN {X 0,Y 534.243,Z 863.938,A -85,B 0,C 180,E1 -837.897,E2 -837.897} C_VEL
LIN {X 0,Y 535.321,Z 843.801,A -85,B 0,C 180,E1 -839.175,E2 -839.175} C_VEL
LIN {X 0,Y 536.394,Z 822.663,A -85,B 0,C 180,E1 -840.279,E2 -840.279} C_VEL
LIN {X 0,Y 537.288,Z 801.75,A -85,B 0,C 180,E1 -841.154,E2 -841.154} C_VEL
LIN {X 0,Y 538.052,Z 779.811,A -85,B 0,C 180,E1 -841.854,E2 -841.854} C_VEL
LIN {X 0,Y 538.609,Z 757.854,A -85,B 0,C 180,E1 -842.344,E2 -842.344} C_VEL
LIN {X 0,Y 539.718,Z 666.089,A -85,B 0,C 180,E1 -843.744,E2 -843.744} C_VEL
LIN {X 0,Y 541.823,Z 658.169,A -85,B 0,C 180,E1 -844.076,E2 -844.076} C_VEL
LIN {X 0,Y 544.956,Z 642.744,A -85,B 0,C 180,E1 -844.437,E2 -844.437} C_VEL
LIN {X 0,Y 547.732,Z 621.552,A -85,B 0,C 180,E1 -844.758,E2 -844.758} C_VEL
LIN {X 0,Y 551.644,Z 574.743,A -85,B 0,C 180,E1 -845.339,E2 -845.339} C_VEL
LIN {X 0,Y 553.42,Z 567.973,A -85,B 0,C 180,E1 -845.598,E2 -845.598} C_VEL
LIN {X 0,Y 556.198,Z 549.758,A -85,B 0,C 180,E1 -845.995,E2 -845.995} C_VEL
LIN {X 0,Y 560.117,Z 514.053,A -85,B 0,C 180,E1 -846.544,E2 -846.544} C_VEL
LIN {X 0,Y 563.673,Z 474.097,A -85,B 0,C 180,E1 -847.028,E2 -847.028} C_VEL
LIN {X 0,Y 563.861,Z 474.035,A -85,B 0,C 180,E1 -847.054,E2 -847.054} C_VEL
LIN {X 0,Y 567.991,Z 485.801,A -85,B 0,C 180,E1 -847.602,E2 -847.602} C_VEL
LIN {X 0,Y 573.062,Z 496.224,A -85,B 0,C 180,E1 -848.256,E2 -848.256} C_VEL
LIN {X 0,Y 579.305,Z 505.544,A -85,B 0,C 180,E1 -849.032,E2 -849.032} C_VEL
LIN {X 0,Y 582.812,Z 510.018,A -85,B 0,C 180,E1 -849.529,E2 -849.529} C_VEL
LIN {X 0,Y 584.631,Z 513.406,A -85,B 0,C 180,E1 -850.083,E2 -850.083} C_VEL
LIN {X 0,Y 584.906,Z 515.978,A -85,B 0,C 180,E1 -850.7,E2 -850.7} C_VEL
LIN {X 0,Y 583.883,Z 517.376,A -85,B 0,C 180,E1 -851.258,E2 -851.258} C_VEL
LIN {X 0,Y 581.392,Z 517.917,A -85,B 0,C 180,E1 -851.871,E2 -851.871} C_VEL
LIN {X 0,Y 578.03,Z 517.344,A -85,B 0,C 180,E1 -852.387,E2 -852.387} C_VEL
LIN {X 0,Y 570.634,Z 514.13,A -85,B 0,C 180,E1 -853.205,E2 -853.205} C_VEL
LIN {X 0,Y 563.071,Z 508.841,A -85,B 0,C 180,E1 -854.161,E2 -854.161} C_VEL
LIN {X 0,Y 556.896,Z 502.162,A -85,B 0,C 180,E1 -855.123,E2 -855.123} C_VEL
LIN {X 0,Y 552.078,Z 494.173,A -85,B 0,C 180,E1 -856.081,E2 -856.081} C_VEL
LIN {X 0,Y 548.448,Z 484.38,A -85,B 0,C 180,E1 -857.085,E2 -857.085} C_VEL
LIN {X 0,Y 546.226,Z 472.337,A -85,B 0,C 180,E1 -858.159,E2 -858.159} C_VEL
LIN {X 0,Y 545.436,Z 458.201,A -85,B 0,C 180,E1 -859.263,E2 -859.263} C_VEL
LIN {X 0,Y 548.05,Z 404.116,A -85,B 0,C 180,E1 -863.042,E2 -863.042} C_VEL
LIN {X 0,Y 548.05,Z 400.707,A -85,B 0,C 180,E1 -863.31,E2 -863.31} C_VEL
LIN {X 0,Y 540.77,Z 387.529,A -85,B 0,C 180,E1 -865.287,E2 -865.287} C_VEL
LIN {X 0,Y 536.086,Z 379.062,A -85,B 0,C 180,E1 -866.619,E2 -866.619} C_VEL
LIN {X 0,Y 533.198,Z 374.029,A -85,B 0,C 180,E1 -867.44,E2 -867.44} C_VEL
LIN {X 0,Y 530.792,Z 369.563,A -85,B 0,C 180,E1 -868.168,E2 -868.168} C_VEL
LIN {X 0,Y 528.926,Z 366.622,A -85,B 0,C 180,E1 -868.698,E2 -868.698} C_VEL
LIN {X 0,Y 528.522,Z 364.902,A -85,B 0,C 180,E1 -868.942,E2 -868.942} C_VEL
LIN {X 0,Y 528.507,Z 364.903,A -85,B 0,C 180,E1 -872.387,E2 -872.387} C_VEL
LIN {X 0,Y 528.522,Z 364.899,A -85,B 0,C 180,E1 -875.763,E2 -875.763} C_VEL
LIN {X 0,Y 528.485,Z 364.903,A -85,B 0,C 180,E1 -879.166,E2 -879.166} C_VEL
LIN {X 0,Y 528.515,Z 364.898,A -85,B 0,C 180,E1 -882.608,E2 -882.608} C_VEL
LIN {X 0,Y 528.494,Z 364.901,A -85,B 0,C 180,E1 -885.986,E2 -885.986} C_VEL
LIN {X 0,Y 528.488,Z 364.905,A -85,B 0,C 180,E1 -889.536,E2 -889.536} C_VEL
LIN {X 0,Y 528.528,Z 364.9,A -85,B 0,C 180,E1 -892.937,E2 -892.937} C_VEL
LIN {X 0,Y 528.507,Z 364.904,A -85,B 0,C 180,E1 -896.421,E2 -896.421} C_VEL
LIN {X 0,Y 528.523,Z 364.904,A -85,B 0,C 180,E1 -899.892,E2 -899.892} C_VEL
LIN {X 0,Y 528.499,Z 364.907,A -85,B 0,C 180,E1 -903.363,E2 -903.363} C_VEL
LIN {X 0,Y 528.515,Z 364.903,A -85,B 0,C 180,E1 -906.683,E2 -906.683} C_VEL
LIN {X 0,Y 528.478,Z 364.904,A -85,B 0,C 180,E1 -910.134,E2 -910.134} C_VEL
LIN {X 0,Y 528.522,Z 364.899,A -85,B 0,C 180,E1 -913.567,E2 -913.567} C_VEL
LIN {X 0,Y 528.479,Z 364.904,A -85,B 0,C 180,E1 -916.826,E2 -916.826} C_VEL
LIN {X 0,Y 528.499,Z 364.902,A -85,B 0,C 180,E1 -920.372,E2 -920.372} C_VEL
LIN {X 0,Y 528.524,Z 364.899,A -85,B 0,C 180,E1 -923.763,E2 -923.763} C_VEL
LIN {X 0,Y 528.508,Z 364.9,A -85,B 0,C 180,E1 -927.247,E2 -927.247} C_VEL
LIN {X 0,Y 528.523,Z 364.9,A -85,B 0,C 180,E1 -930.598,E2 -930.598} C_VEL
LIN {X 0,Y 528.525,Z 364.899,A -85,B 0,C 180,E1 -934.054,E2 -934.054} C_VEL
LIN {X 0,Y 528.506,Z 364.894,A -85,B 0,C 180,E1 -937.53,E2 -937.53} C_VEL
LIN {X 0,Y 528.526,Z 364.894,A -85,B 0,C 180,E1 -938.325,E2 -938.325} C_VEL
LIN {X 0,Y 527.546,Z 365.023,A -85,B 0,C 180,E1 -939.16,E2 -939.16} C_VEL
LIN {X 0,Y 521.1,Z 365.819,A -85,B 0,C 180,E1 -941.505,E2 -941.505} C_VEL
LIN {X 0,Y 520.585,Z 365.876,A -85,B 0,C 180,E1 -942.116,E2 -942.116} C_VEL
LIN {X 0,Y 520.564,Z 365.891,A -85,B 0,C 180,E1 -945.603,E2 -945.603} C_VEL
LIN {X 0,Y 520.553,Z 365.896,A -85,B 0,C 180,E1 -949.082,E2 -949.082} C_VEL
LIN {X 0,Y 520.574,Z 365.891,A -85,B 0,C 180,E1 -952.355,E2 -952.355} C_VEL
LIN {X 0,Y 520.58,Z 366.028,A -85,B 0,C 180,E1 -955.22,E2 -955.22} C_VEL
LIN {X 0,Y 528.691,Z 387.671,A -85,B 0,C 180,E1 -957.409,E2 -957.409} C_VEL
LIN {X 0,Y 527.81,Z 420.991,A -85,B 0,C 180,E1 -959.93,E2 -959.93} C_VEL
LIN {X 0,Y 526.577,Z 467.331,A -85,B 0,C 180,E1 -963.317,E2 -963.317} C_VEL
LIN {X 0,Y 526.524,Z 478.032,A -85,B 0,C 180,E1 -964.041,E2 -964.041} C_VEL
LIN {X 0,Y 527.555,Z 486.496,A -85,B 0,C 180,E1 -964.225,E2 -964.225} C_VEL
LIN {X 0,Y 525.896,Z 685.003,A -85,B 0,C 180,E1 -967.105,E2 -967.105} C_VEL
LIN {X 0,Y 525.552,Z 703.391,A -85,B 0,C 180,E1 -967.566,E2 -967.566} C_VEL
LIN {X 0,Y 525.058,Z 720.936,A -85,B 0,C 180,E1 -968.202,E2 -968.202} C_VEL
LIN {X 0,Y 524.446,Z 737.48,A -85,B 0,C 180,E1 -968.997,E2 -968.997} C_VEL
LIN {X 0,Y 523.752,Z 753.381,A -85,B 0,C 180,E1 -969.961,E2 -969.961} C_VEL
LIN {X 0,Y 523.02,Z 769.257,A -85,B 0,C 180,E1 -971.151,E2 -971.151} C_VEL
LIN {X 0,Y 522.288,Z 783.316,A -85,B 0,C 180,E1 -972.434,E2 -972.434} C_VEL
LIN {X 0,Y 521.609,Z 796.362,A -85,B 0,C 180,E1 -973.863,E2 -973.863} C_VEL
LIN {X 0,Y 521.003,Z 810.367,A -85,B 0,C 180,E1 -975.667,E2 -975.667} C_VEL
LIN {X 0,Y 520.573,Z 821.863,A -85,B 0,C 180,E1 -977.465,E2 -977.465} C_VEL
LIN {X 0,Y 520.267,Z 831.786,A -85,B 0,C 180,E1 -979.369,E2 -979.369} C_VEL
LIN {X 0,Y 520.078,Z 839.717,A -85,B 0,C 180,E1 -981.264,E2 -981.264} C_VEL
LIN {X 0,Y 519.975,Z 846.193,A -85,B 0,C 180,E1 -983.264,E2 -983.264} C_VEL
LIN {X 0,Y 519.926,Z 850.883,A -85,B 0,C 180,E1 -985.257,E2 -985.257} C_VEL
LIN {X 0,Y 519.909,Z 853.907,A -85,B 0,C 180,E1 -987.245,E2 -987.245} C_VEL
LIN {X 0,Y 519.913,Z 855.34,A -85,B 0,C 180,E1 -989.229,E2 -989.229} C_VEL
LIN {X 0,Y 519.907,Z 855.211,A -85,B 0,C 180,E1 -991.212,E2 -991.212} C_VEL
LIN {X 0,Y 519.913,Z 853.515,A -85,B 0,C 180,E1 -993.197,E2 -993.197} C_VEL
LIN {X 0,Y 519.93,Z 849.96,A -85,B 0,C 180,E1 -995.297,E2 -995.297} C_VEL
LIN {X 0,Y 519.988,Z 844.862,A -85,B 0,C 180,E1 -997.291,E2 -997.291} C_VEL
LIN {X 0,Y 520.122,Z 837.93,A -85,B 0,C 180,E1 -999.293,E2 -999.293} C_VEL
LIN {X 0,Y 520.331,Z 829.523,A -85,B 0,C 180,E1 -1001.191,E2 -1001.191} C_VEL
LIN {X 0,Y 520.65,Z 819.71,A -85,B 0,C 180,E1 -1002.985,E2 -1002.985} C_VEL
LIN {X 0,Y 521.089,Z 808.012,A -85,B 0,C 180,E1 -1004.744,E2 -1004.744} C_VEL
LIN {X 0,Y 521.826,Z 792.319,A -85,B 0,C 180,E1 -1006.703,E2 -1006.703} C_VEL
LIN {X 0,Y 522.576,Z 778.017,A -85,B 0,C 180,E1 -1008.172,E2 -1008.172} C_VEL
LIN {X 0,Y 523.356,Z 762.54,A -85,B 0,C 180,E1 -1009.474,E2 -1009.474} C_VEL
LIN {X 0,Y 524.062,Z 746.359,A -85,B 0,C 180,E1 -1010.583,E2 -1010.583} C_VEL
LIN {X 0,Y 524.736,Z 730.383,A -85,B 0,C 180,E1 -1011.46,E2 -1011.46} C_VEL
LIN {X 0,Y 525.317,Z 712.655,A -85,B 0,C 180,E1 -1012.213,E2 -1012.213} C_VEL
LIN {X 0,Y 525.741,Z 694.449,A -85,B 0,C 180,E1 -1012.774,E2 -1012.774} C_VEL
LIN {X 0,Y 526.011,Z 675.07,A -85,B 0,C 180,E1 -1013.156,E2 -1013.156} C_VEL
LIN {X 0,Y 527.412,Z 483.763,A -85,B 0,C 180,E1 -1015.914,E2 -1015.914} C_VEL
LIN {X 0,Y 526.371,Z 476.792,A -85,B 0,C 180,E1 -1016.094,E2 -1016.094} C_VEL
LIN {X 0,Y 527.588,Z 428.78,A -85,B 0,C 180,E1 -1019.584,E2 -1019.584} C_VEL
LIN {X 0,Y 528.797,Z 388.115,A -85,B 0,C 180,E1 -1022.641,E2 -1022.641} C_VEL
LIN {X 0,Y 522.756,Z 371.989,A -85,B 0,C 180,E1 -1024.282,E2 -1024.282} C_VEL
LIN {X 0,Y 520.583,Z 365.884,A -85,B 0,C 180,E1 -1024.903,E2 -1024.903} C_VEL
LIN {X 0,Y 520.527,Z 365.895,A -85,B 0,C 180,E1 -1028.22,E2 -1028.22} C_VEL
LIN {X 0,Y 520.556,Z 365.891,A -85,B 0,C 180,E1 -1031.654,E2 -1031.654} C_VEL
LIN {X 0,Y 520.55,Z 365.883,A -85,B 0,C 180,E1 -1034.865,E2 -1034.865} C_VEL
LIN {X 0,Y 520.531,Z 365.885,A -85,B 0,C 180,E1 -1038.2,E2 -1038.2} C_VEL
LIN {X 0,Y 520.586,Z 365.881,A -85,B 0,C 180,E1 -1041.516,E2 -1041.516} C_VEL
LIN {X 0,Y 520.535,Z 365.954,A -85,B 0,C 180,E1 -1042.458,E2 -1042.458} C_VEL
LIN {X 0,Y 521.801,Z 369.324,A -85,B 0,C 180,E1 -1042.872,E2 -1042.872} C_VEL
LIN {X 0,Y 529.912,Z 389.796,A -85,B 0,C 180,E1 -1045.353,E2 -1045.353} C_VEL
LIN {X 0,Y 530.57,Z 391.737,A -85,B 0,C 180,E1 -1045.573,E2 -1045.573} C_VEL
LIN {X 0,Y 529.06,Z 431.38,A -85,B 0,C 180,E1 -1048.813,E2 -1048.813} C_VEL
LIN {X 0,Y 527.355,Z 474.206,A -85,B 0,C 180,E1 -1052.259,E2 -1052.259} C_VEL
LIN {X 0,Y 525.739,Z 519.024,A -85,B 0,C 180,E1 -1055.805,E2 -1055.805} C_VEL
LIN {X 0,Y 524.251,Z 564.215,A -85,B 0,C 180,E1 -1059.339,E2 -1059.339} C_VEL
LIN {X 0,Y 523.569,Z 591.691,A -85,B 0,C 180,E1 -1061.43,E2 -1061.43} C_VEL
LIN {X 0,Y 524.157,Z 599.879,A -85,B 0,C 180,E1 -1061.589,E2 -1061.589} C_VEL
LIN {X 0,Y 523.547,Z 674.577,A -85,B 0,C 180,E1 -1062.677,E2 -1062.677} C_VEL
LIN {X 0,Y 523.032,Z 735.572,A -85,B 0,C 180,E1 -1063.615,E2 -1063.615} C_VEL
LIN {X 0,Y 522.776,Z 752.348,A -85,B 0,C 180,E1 -1064.098,E2 -1064.098} C_VEL
LIN {X 0,Y 522.478,Z 766.391,A -85,B 0,C 180,E1 -1064.688,E2 -1064.688} C_VEL
LIN {X 0,Y 522.069,Z 781.387,A -85,B 0,C 180,E1 -1065.526,E2 -1065.526} C_VEL
LIN {X 0,Y 521.642,Z 794.441,A -85,B 0,C 180,E1 -1066.476,E2 -1066.476} C_VEL
LIN {X 0,Y 521.259,Z 805.971,A -85,B 0,C 180,E1 -1067.514,E2 -1067.514} C_VEL
LIN {X 0,Y 520.857,Z 817.76,A -85,B 0,C 180,E1 -1068.82,E2 -1068.82} C_VEL
LIN {X 0,Y 520.534,Z 827.589,A -85,B 0,C 180,E1 -1070.195,E2 -1070.195} C_VEL
LIN {X 0,Y 520.322,Z 835.143,A -85,B 0,C 180,E1 -1071.491,E2 -1071.491} C_VEL
LIN {X 0,Y 520.133,Z 842.434,A -85,B 0,C 180,E1 -1073.044,E2 -1073.044} C_VEL
LIN {X 0,Y 520.013,Z 848.213,A -85,B 0,C 180,E1 -1074.704,E2 -1074.704} C_VEL
LIN {X 0,Y 519.96,Z 852.072,A -85,B 0,C 180,E1 -1076.251,E2 -1076.251} C_VEL
LIN {X 0,Y 519.937,Z 854.758,A -85,B 0,C 180,E1 -1077.906,E2 -1077.906} C_VEL
LIN {X 0,Y 519.932,Z 855.942,A -85,B 0,C 180,E1 -1079.834,E2 -1079.834} C_VEL
LIN {X 0,Y 519.936,Z 855.46,A -85,B 0,C 180,E1 -1081.432,E2 -1081.432} C_VEL
LIN {X 0,Y 519.958,Z 853.447,A -85,B 0,C 180,E1 -1083.196,E2 -1083.196} C_VEL
LIN {X 0,Y 520.018,Z 849.583,A -85,B 0,C 180,E1 -1084.963,E2 -1084.963} C_VEL
LIN {X 0,Y 520.124,Z 844.713,A -85,B 0,C 180,E1 -1086.512,E2 -1086.512} C_VEL
LIN {X 0,Y 520.331,Z 837.765,A -85,B 0,C 180,E1 -1088.175,E2 -1088.175} C_VEL
LIN {X 0,Y 520.594,Z 829.204,A -85,B 0,C 180,E1 -1089.73,E2 -1089.73} C_VEL
LIN {X 0,Y 520.923,Z 820.072,A -85,B 0,C 180,E1 -1091.066,E2 -1091.066} C_VEL
LIN {X 0,Y 521.396,Z 807.591,A -85,B 0,C 180,E1 -1092.515,E2 -1092.515} C_VEL
LIN {X 0,Y 521.841,Z 795.458,A -85,B 0,C 180,E1 -1093.631,E2 -1093.631} C_VEL
LIN {X 0,Y 522.325,Z 780.838,A -85,B 0,C 180,E1 -1094.693,E2 -1094.693} C_VEL
LIN {X 0,Y 522.709,Z 766.631,A -85,B 0,C 180,E1 -1095.476,E2 -1095.476} C_VEL
LIN {X 0,Y 523.012,Z 750.519,A -85,B 0,C 180,E1 -1096.129,E2 -1096.129} C_VEL
LIN {X 0,Y 523.197,Z 734.61,A -85,B 0,C 180,E1 -1096.549,E2 -1096.549} C_VEL
LIN {X 0,Y 524.917,Z 617.664,A -85,B 0,C 180,E1 -1098.468,E2 -1098.468} C_VEL
LIN {X 0,Y 525.4,Z 597.039,A -85,B 0,C 180,E1 -1098.847,E2 -1098.847} C_VEL
LIN {X 0,Y 527.334,Z 566.935,A -85,B 0,C 180,E1 -1101.348,E2 -1101.348} C_VEL
LIN {X 0,Y 530.18,Z 529.372,A -85,B 0,C 180,E1 -1104.572,E2 -1104.572} C_VEL
LIN {X 0,Y 534.354,Z 489.729,A -85,B 0,C 180,E1 -1108.133,E2 -1108.133} C_VEL
LIN {X 0,Y 538.695,Z 460.07,A -85,B 0,C 180,E1 -1110.961,E2 -1110.961} C_VEL
LIN {X 0,Y 543.912,Z 435.462,A -85,B 0,C 180,E1 -1113.468,E2 -1113.468} C_VEL
LIN {X 0,Y 549.191,Z 418.352,A -85,B 0,C 180,E1 -1115.376,E2 -1115.376} C_VEL
LIN {X 0,Y 550.138,Z 415.649,A -85,B 0,C 180,E1 -1115.754,E2 -1115.754} C_VEL
LIN {X 0,Y 550.07,Z 414.049,A -85,B 0,C 180,E1 -1116.598,E2 -1116.598} C_VEL
LIN {X 0,Y 550.049,Z 413.921,A -85,B 0,C 180,E1 -1116.791,E2 -1116.791} C_VEL
LIN {X 0,Y 543.724,Z 425.403,A -85,B 0,C 180,E1 -1117.917,E2 -1117.917} C_VEL
LIN {X 0,Y 538.96,Z 438.36,A -85,B 0,C 180,E1 -1119.077,E2 -1119.077} C_VEL
LIN {X 0,Y 536.057,Z 452.419,A -85,B 0,C 180,E1 -1120.281,E2 -1120.281} C_VEL
LIN {X 0,Y 535.259,Z 466.54,A -85,B 0,C 180,E1 -1121.49,E2 -1121.49} C_VEL
LIN {X 0,Y 536.59,Z 479.147,A -85,B 0,C 180,E1 -1122.605,E2 -1122.605} C_VEL
LIN {X 0,Y 539.708,Z 490.203,A -85,B 0,C 180,E1 -1123.637,E2 -1123.637} C_VEL
LIN {X 0,Y 544.296,Z 499.535,A -85,B 0,C 180,E1 -1124.565,E2 -1124.565} C_VEL
LIN {X 0,Y 550.879,Z 508.324,A -85,B 0,C 180,E1 -1125.504,E2 -1125.504} C_VEL
LIN {X 0,Y 558.496,Z 515.398,A -85,B 0,C 180,E1 -1126.325,E2 -1126.325} C_VEL
LIN {X 0,Y 567.581,Z 521.349,A -85,B 0,C 180,E1 -1127.124,E2 -1127.124} C_VEL
LIN {X 0,Y 572.969,Z 523.89,A -85,B 0,C 180,E1 -1127.574,E2 -1127.574} C_VEL
LIN {X 0,Y 576.886,Z 525.014,A -85,B 0,C 180,E1 -1128.034,E2 -1128.034} C_VEL
LIN {X 0,Y 580.035,Z 525.151,A -85,B 0,C 180,E1 -1128.577,E2 -1128.577} C_VEL
LIN {X 0,Y 581.928,Z 524.395,A -85,B 0,C 180,E1 -1129.112,E2 -1129.112} C_VEL
LIN {X 0,Y 582.759,Z 522.578,A -85,B 0,C 180,E1 -1129.735,E2 -1129.735} C_VEL
LIN {X 0,Y 582.07,Z 519.778,A -85,B 0,C 180,E1 -1130.339,E2 -1130.339} C_VEL
LIN {X 0,Y 579.872,Z 516.298,A -85,B 0,C 180,E1 -1130.869,E2 -1130.869} C_VEL
LIN {X 0,Y 573.685,Z 508.389,A -85,B 0,C 180,E1 -1131.666,E2 -1131.666} C_VEL
LIN {X 0,Y 567.919,Z 498.834,A -85,B 0,C 180,E1 -1132.407,E2 -1132.407} C_VEL
LIN {X 0,Y 566.596,Z 496.473,A -85,B 0,C 180,E1 -1132.581,E2 -1132.581} C_VEL
LIN {X 0,Y 562.324,Z 539.289,A -85,B 0,C 180,E1 -1133.154,E2 -1133.154} C_VEL
LIN {X 0,Y 558.859,Z 565.064,A -85,B 0,C 180,E1 -1133.631,E2 -1133.631} C_VEL
LIN {X 0,Y 556.569,Z 576.04,A -85,B 0,C 180,E1 -1133.952,E2 -1133.952} C_VEL
LIN {X 0,Y 555.899,Z 578.96,A -85,B 0,C 180,E1 -1134.047,E2 -1134.047} C_VEL
LIN {X 0,Y 552.925,Z 612.03,A -85,B 0,C 180,E1 -1134.407,E2 -1134.407} C_VEL
LIN {X 0,Y 548.978,Z 634.986,A -85,B 0,C 180,E1 -1134.635,E2 -1134.635} C_VEL
LIN {X 0,Y 544.488,Z 653.611,A -85,B 0,C 180,E1 -1134.94,E2 -1134.94} C_VEL
LIN {X 0,Y 541.239,Z 665.725,A -85,B 0,C 180,E1 -1135.304,E2 -1135.304} C_VEL
LIN {X 0,Y 540.024,Z 670.223,A -85,B 0,C 180,E1 -1135.482,E2 -1135.482} C_VEL
LIN {X 0,Y 536.036,Z 684.51,A -85,B 0,C 180,E1 -1135.771,E2 -1135.771} C_VEL
LIN {X 0,Y 533.169,Z 695.011,A -85,B 0,C 180,E1 -1136.153,E2 -1136.153} C_VEL
LIN {X 0,Y 532.572,Z 698.239,A -85,B 0,C 180,E1 -1136.283,E2 -1136.283} C_VEL
LIN {X 0,Y 531.758,Z 762.198,A -85,B 0,C 180,E1 -1137.276,E2 -1137.276} C_VEL
LIN {X 0,Y 531.068,Z 783.863,A -85,B 0,C 180,E1 -1137.804,E2 -1137.804} C_VEL
LIN {X 0,Y 530.194,Z 806.299,A -85,B 0,C 180,E1 -1138.571,E2 -1138.571} C_VEL
LIN {X 0,Y 529.157,Z 827.27,A -85,B 0,C 180,E1 -1139.499,E2 -1139.499} C_VEL
LIN {X 0,Y 528.008,Z 847.793,A -85,B 0,C 180,E1 -1140.629,E2 -1140.629} C_VEL
LIN {X 0,Y 526.773,Z 867.707,A -85,B 0,C 180,E1 -1141.958,E2 -1141.958} C_VEL
LIN {X 0,Y 525.528,Z 887.134,A -85,B 0,C 180,E1 -1143.502,E2 -1143.502} C_VEL
LIN {X 0,Y 524.353,Z 905.27,A -85,B 0,C 180,E1 -1145.196,E2 -1145.196} C_VEL
LIN {X 0,Y 523.196,Z 923.219,A -85,B 0,C 180,E1 -1147.173,E2 -1147.173} C_VEL
LIN {X 0,Y 522.227,Z 939.283,A -85,B 0,C 180,E1 -1149.255,E2 -1149.255} C_VEL
LIN {X 0,Y 521.439,Z 953.602,A -85,B 0,C 180,E1 -1151.439,E2 -1151.439} C_VEL
LIN {X 0,Y 520.835,Z 966.276,A -85,B 0,C 180,E1 -1153.723,E2 -1153.723} C_VEL
LIN {X 0,Y 520.433,Z 976.858,A -85,B 0,C 180,E1 -1155.991,E2 -1155.991} C_VEL
LIN {X 0,Y 520.165,Z 985.921,A -85,B 0,C 180,E1 -1158.356,E2 -1158.356} C_VEL
LIN {X 0,Y 520.015,Z 993.099,A -85,B 0,C 180,E1 -1160.705,E2 -1160.705} C_VEL
LIN {X 0,Y 519.942,Z 998.594,A -85,B 0,C 180,E1 -1163.041,E2 -1163.041} C_VEL
LIN {X 0,Y 519.917,Z 1002.585,A -85,B 0,C 180,E1 -1165.477,E2 -1165.477} C_VEL
LIN {X 0,Y 519.912,Z 1004.836,A -85,B 0,C 180,E1 -1167.906,E2 -1167.906} C_VEL
LIN {X 0,Y 519.894,Z 1005.447,A -85,B 0,C 180,E1 -1170.44,E2 -1170.44} C_VEL
LIN {X 0,Y 519.894,Z 1004.329,A -85,B 0,C 180,E1 -1172.866,E2 -1172.866} C_VEL
LIN {X 0,Y 519.903,Z 1001.651,A -85,B 0,C 180,E1 -1175.186,E2 -1175.186} C_VEL
LIN {X 0,Y 519.949,Z 997.197,A -85,B 0,C 180,E1 -1177.625,E2 -1177.625} C_VEL
LIN {X 0,Y 520.044,Z 991.251,A -85,B 0,C 180,E1 -1179.964,E2 -1179.964} C_VEL
LIN {X 0,Y 520.231,Z 983.512,A -85,B 0,C 180,E1 -1182.318,E2 -1182.318} C_VEL
LIN {X 0,Y 520.551,Z 973.879,A -85,B 0,C 180,E1 -1184.687,E2 -1184.687} C_VEL
LIN {X 0,Y 521.015,Z 962.746,A -85,B 0,C 180,E1 -1186.959,E2 -1186.959} C_VEL
LIN {X 0,Y 521.668,Z 949.348,A -85,B 0,C 180,E1 -1189.248,E2 -1189.248} C_VEL
LIN {X 0,Y 522.467,Z 935.055,A -85,B 0,C 180,E1 -1191.322,E2 -1191.322} C_VEL
LIN {X 0,Y 523.471,Z 918.728,A -85,B 0,C 180,E1 -1193.349,E2 -1193.349} C_VEL
LIN {X 0,Y 524.604,Z 901.15,A -85,B 0,C 180,E1 -1195.212,E2 -1195.212} C_VEL
LIN {X 0,Y 525.807,Z 883.05,A -85,B 0,C 180,E1 -1196.848,E2 -1196.848} C_VEL
LIN {X 0,Y 527.039,Z 863.741,A -85,B 0,C 180,E1 -1198.326,E2 -1198.326} C_VEL
LIN {X 0,Y 528.214,Z 843.8,A -85,B 0,C 180,E1 -1199.607,E2 -1199.607} C_VEL
LIN {X 0,Y 529.415,Z 822.535,A -85,B 0,C 180,E1 -1200.728,E2 -1200.728} C_VEL
LIN {X 0,Y 530.422,Z 800.983,A -85,B 0,C 180,E1 -1201.635,E2 -1201.635} C_VEL
LIN {X 0,Y 531.275,Z 778.859,A -85,B 0,C 180,E1 -1202.338,E2 -1202.338} C_VEL
LIN {X 0,Y 531.862,Z 756.802,A -85,B 0,C 180,E1 -1202.825,E2 -1202.825} C_VEL
LIN {X 0,Y 532.681,Z 696.923,A -85,B 0,C 180,E1 -1203.752,E2 -1203.752} C_VEL
LIN {X 0,Y 535.531,Z 686.308,A -85,B 0,C 180,E1 -1204.176,E2 -1204.176} C_VEL
LIN {X 0,Y 539.481,Z 672.226,A -85,B 0,C 180,E1 -1204.49,E2 -1204.49} C_VEL
LIN {X 0,Y 540.528,Z 668.349,A -85,B 0,C 180,E1 -1204.576,E2 -1204.576} C_VEL
LIN {X 0,Y 543.235,Z 658.333,A -85,B 0,C 180,E1 -1204.943,E2 -1204.943} C_VEL
LIN {X 0,Y 547.513,Z 641.508,A -85,B 0,C 180,E1 -1205.279,E2 -1205.279} C_VEL
LIN {X 0,Y 551.793,Z 619.884,A -85,B 0,C 180,E1 -1205.519,E2 -1205.519} C_VEL
LIN {X 0,Y 554.55,Z 596.368,A -85,B 0,C 180,E1 -1205.76,E2 -1205.76} C_VEL
LIN {X 0,Y 556.162,Z 577.387,A -85,B 0,C 180,E1 -1205.99,E2 -1205.99} C_VEL
LIN {X 0,Y 558.318,Z 568.164,A -85,B 0,C 180,E1 -1206.294,E2 -1206.294} C_VEL
LIN {X 0,Y 561.442,Z 546.658,A -85,B 0,C 180,E1 -1206.725,E2 -1206.725} C_VEL
LIN {X 0,Y 565.569,Z 507.84,A -85,B 0,C 180,E1 -1207.282,E2 -1207.282} C_VEL
LIN {X 0,Y 566.698,Z 496.398,A -85,B 0,C 180,E1 -1207.432,E2 -1207.432} C_VEL
LIN {X 0,Y 572.365,Z 506.452,A -85,B 0,C 180,E1 -1208.167,E2 -1208.167} C_VEL
LIN {X 0,Y 578.898,Z 515.08,A -85,B 0,C 180,E1 -1208.985,E2 -1208.985} C_VEL
LIN {X 0,Y 581.496,Z 518.686,A -85,B 0,C 180,E1 -1209.474,E2 -1209.474} C_VEL
LIN {X 0,Y 582.709,Z 521.784,A -85,B 0,C 180,E1 -1210.068,E2 -1210.068} C_VEL
LIN {X 0,Y 582.428,Z 523.801,A -85,B 0,C 180,E1 -1210.643,E2 -1210.643} C_VEL
LIN {X 0,Y 580.755,Z 525,A -85,B 0,C 180,E1 -1211.253,E2 -1211.253} C_VEL
LIN {X 0,Y 578.026,Z 525.173,A -85,B 0,C 180,E1 -1211.795,E2 -1211.795} C_VEL
LIN {X 0,Y 574.356,Z 524.372,A -85,B 0,C 180,E1 -1212.281,E2 -1212.281} C_VEL
LIN {X 0,Y 565.481,Z 520.369,A -85,B 0,C 180,E1 -1213.241,E2 -1213.241} C_VEL
LIN {X 0,Y 557.364,Z 514.452,A -85,B 0,C 180,E1 -1214.294,E2 -1214.294} C_VEL
LIN {X 0,Y 550.647,Z 506.826,A -85,B 0,C 180,E1 -1215.38,E2 -1215.38} C_VEL
LIN {X 0,Y 545.585,Z 497.876,A -85,B 0,C 180,E1 -1216.444,E2 -1216.444} C_VEL
LIN {X 0,Y 542.123,Z 487.803,A -85,B 0,C 180,E1 -1217.472,E2 -1217.472} C_VEL
LIN {X 0,Y 539.952,Z 474.998,A -85,B 0,C 180,E1 -1218.618,E2 -1218.618} C_VEL
LIN {X 0,Y 539.315,Z 459.861,A -85,B 0,C 180,E1 -1219.802,E2 -1219.802} C_VEL
LIN {X 0,Y 542.135,Z 408.288,A -85,B 0,C 180,E1 -1223.437,E2 -1223.437} C_VEL
LIN {X 0,Y 542.27,Z 405.483,A -85,B 0,C 180,E1 -1223.645,E2 -1223.645} C_VEL
LIN {X 0,Y 533.602,Z 389.671,A -85,B 0,C 180,E1 -1226.056,E2 -1226.056} C_VEL
LIN {X 0,Y 527.813,Z 379.541,A -85,B 0,C 180,E1 -1227.71,E2 -1227.71} C_VEL
LIN {X 0,Y 525.386,Z 375.171,A -85,B 0,C 180,E1 -1228.443,E2 -1228.443} C_VEL
LIN {X 0,Y 523.373,Z 371.275,A -85,B 0,C 180,E1 -1229.076,E2 -1229.076} C_VEL
LIN {X 0,Y 521.152,Z 368.028,A -85,B 0,C 180,E1 -1229.697,E2 -1229.697} C_VEL
LIN {X 0,Y 520.592,Z 365.887,A -85,B 0,C 180,E1 -1230.019,E2 -1230.019} C_VEL
LIN {X 0,Y 520.546,Z 365.895,A -85,B 0,C 180,E1 -1233.414,E2 -1233.414} C_VEL
LIN {X 0,Y 520.583,Z 365.89,A -85,B 0,C 180,E1 -1236.924,E2 -1236.924} C_VEL
LIN {X 0,Y 520.574,Z 365.89,A -85,B 0,C 180,E1 -1240.36,E2 -1240.36} C_VEL
LIN {X 0,Y 520.581,Z 365.888,A -85,B 0,C 180,E1 -1243.83,E2 -1243.83} C_VEL
LIN {X 0,Y 520.549,Z 365.894,A -85,B 0,C 180,E1 -1247.239,E2 -1247.239} C_VEL
LIN {X 0,Y 520.585,Z 365.889,A -85,B 0,C 180,E1 -1250.716,E2 -1250.716} C_VEL
LIN {X 0,Y 520.545,Z 365.891,A -85,B 0,C 180,E1 -1254.047,E2 -1254.047} C_VEL
LIN {X 0,Y 520.558,Z 365.893,A -85,B 0,C 180,E1 -1257.578,E2 -1257.578} C_VEL
LIN {X 0,Y 520.584,Z 365.889,A -85,B 0,C 180,E1 -1260.991,E2 -1260.991} C_VEL
LIN {X 0,Y 520.572,Z 365.896,A -85,B 0,C 180,E1 -1264.56,E2 -1264.56} C_VEL
LIN {X 0,Y 520.586,Z 365.892,A -85,B 0,C 180,E1 -1267.949,E2 -1267.949} C_VEL
LIN {X 0,Y 520.581,Z 365.892,A -85,B 0,C 180,E1 -1271.41,E2 -1271.41} C_VEL
LIN {X 0,Y 520.571,Z 365.889,A -85,B 0,C 180,E1 -1274.801,E2 -1274.801} C_VEL
LIN {X 0,Y 520.541,Z 365.892,A -85,B 0,C 180,E1 -1278.246,E2 -1278.246} C_VEL
LIN {X 0,Y 520.586,Z 365.887,A -85,B 0,C 180,E1 -1281.64,E2 -1281.64} C_VEL
LIN {X 0,Y 520.536,Z 365.893,A -85,B 0,C 180,E1 -1284.998,E2 -1284.998} C_VEL
LIN {X 0,Y 520.569,Z 365.888,A -85,B 0,C 180,E1 -1288.572,E2 -1288.572} C_VEL
LIN {X 0,Y 520.572,Z 365.886,A -85,B 0,C 180,E1 -1291.903,E2 -1291.903} C_VEL
LIN {X 0,Y 520.569,Z 365.881,A -85,B 0,C 180,E1 -1295.32,E2 -1295.32} C_VEL
LIN {X 0,Y 520.588,Z 365.888,A -85,B 0,C 180,E1 -1298.765,E2 -1298.765} C_VEL
LIN {X 0,Y 520.585,Z 365.876,A -85,B 0,C 180,E1 -1302.116,E2 -1302.116} C_VEL
LIN {X 0,Y 519.614,Z 366,A -85,B 0,C 180,E1 -1302.964,E2 -1302.964} C_VEL
LIN {X 0,Y 513.149,Z 366.818,A -85,B 0,C 180,E1 -1305.346,E2 -1305.346} C_VEL
LIN {X 0,Y 512.62,Z 366.878,A -85,B 0,C 180,E1 -1305.967,E2 -1305.967} C_VEL
LIN {X 0,Y 512.61,Z 366.886,A -85,B 0,C 180,E1 -1309.527,E2 -1309.527} C_VEL
LIN {X 0,Y 512.649,Z 366.88,A -85,B 0,C 180,E1 -1312.939,E2 -1312.939} C_VEL
LIN {X 0,Y 512.645,Z 366.953,A -85,B 0,C 180,E1 -1314.704,E2 -1314.704} C_VEL
LIN {X 0,Y 521.293,Z 389.77,A -85,B 0,C 180,E1 -1317.05,E2 -1317.05} C_VEL
LIN {X 0,Y 521.684,Z 392.46,A -85,B 0,C 180,E1 -1317.287,E2 -1317.287} C_VEL
LIN {X 0,Y 520.17,Z 436.865,A -85,B 0,C 180,E1 -1320.65,E2 -1320.65} C_VEL
LIN {X 0,Y 519.284,Z 476.031,A -85,B 0,C 180,E1 -1323.468,E2 -1323.468} C_VEL
LIN {X 0,Y 519.417,Z 479.413,A -85,B 0,C 180,E1 -1323.662,E2 -1323.662} C_VEL
LIN {X 0,Y 520.406,Z 487.664,A -85,B 0,C 180,E1 -1323.844,E2 -1323.844} C_VEL
LIN {X 0,Y 518.581,Z 686.154,A -85,B 0,C 180,E1 -1326.764,E2 -1326.764} C_VEL
LIN {X 0,Y 518.236,Z 704.609,A -85,B 0,C 180,E1 -1327.232,E2 -1327.232} C_VEL
LIN {X 0,Y 517.721,Z 722.159,A -85,B 0,C 180,E1 -1327.877,E2 -1327.877} C_VEL
LIN {X 0,Y 517.074,Z 738.716,A -85,B 0,C 180,E1 -1328.683,E2 -1328.683} C_VEL
LIN {X 0,Y 516.335,Z 754.627,A -85,B 0,C 180,E1 -1329.66,E2 -1329.66} C_VEL
LIN {X 0,Y 515.546,Z 770.508,A -85,B 0,C 180,E1 -1330.867,E2 -1330.867} C_VEL
LIN {X 0,Y 514.743,Z 784.755,A -85,B 0,C 180,E1 -1332.186,E2 -1332.186} C_VEL
LIN {X 0,Y 514.008,Z 797.624,A -85,B 0,C 180,E1 -1333.617,E2 -1333.617} C_VEL
LIN {X 0,Y 513.336,Z 809.634,A -85,B 0,C 180,E1 -1335.217,E2 -1335.217} C_VEL
LIN {X 0,Y 512.784,Z 820.287,A -85,B 0,C 180,E1 -1336.928,E2 -1336.928} C_VEL
LIN {X 0,Y 512.349,Z 830.869,A -85,B 0,C 180,E1 -1338.997,E2 -1338.997} C_VEL
LIN {X 0,Y 512.111,Z 839.318,A -85,B 0,C 180,E1 -1341.014,E2 -1341.014} C_VEL
LIN {X 0,Y 511.987,Z 845.894,A -85,B 0,C 180,E1 -1343.046,E2 -1343.046} C_VEL
LIN {X 0,Y 511.928,Z 850.68,A -85,B 0,C 180,E1 -1345.07,E2 -1345.07} C_VEL
LIN {X 0,Y 511.912,Z 853.795,A -85,B 0,C 180,E1 -1347.089,E2 -1347.089} C_VEL
LIN {X 0,Y 511.91,Z 855.318,A -85,B 0,C 180,E1 -1349.105,E2 -1349.105} C_VEL
LIN {X 0,Y 511.907,Z 855.211,A -85,B 0,C 180,E1 -1351.231,E2 -1351.231} C_VEL
LIN {X 0,Y 511.914,Z 853.515,A -85,B 0,C 180,E1 -1353.247,E2 -1353.247} C_VEL
LIN {X 0,Y 511.934,Z 849.958,A -85,B 0,C 180,E1 -1355.38,E2 -1355.38} C_VEL
LIN {X 0,Y 511.999,Z 844.859,A -85,B 0,C 180,E1 -1357.406,E2 -1357.406} C_VEL
LIN {X 0,Y 512.147,Z 837.926,A -85,B 0,C 180,E1 -1359.439,E2 -1359.439} C_VEL
LIN {X 0,Y 512.388,Z 829.517,A -85,B 0,C 180,E1 -1361.367,E2 -1361.367} C_VEL
LIN {X 0,Y 512.842,Z 819.056,A -85,B 0,C 180,E1 -1363.375,E2 -1363.375} C_VEL
LIN {X 0,Y 513.429,Z 807.86,A -85,B 0,C 180,E1 -1365.127,E2 -1365.127} C_VEL
LIN {X 0,Y 514.127,Z 795.487,A -85,B 0,C 180,E1 -1366.728,E2 -1366.728} C_VEL
LIN {X 0,Y 514.918,Z 781.603,A -85,B 0,C 180,E1 -1368.218,E2 -1368.218} C_VEL
LIN {X 0,Y 515.748,Z 766.685,A -85,B 0,C 180,E1 -1369.538,E2 -1369.538} C_VEL
LIN {X 0,Y 516.518,Z 750.794,A -85,B 0,C 180,E1 -1370.688,E2 -1370.688} C_VEL
LIN {X 0,Y 517.297,Z 733.902,A -85,B 0,C 180,E1 -1371.665,E2 -1371.665} C_VEL
LIN {X 0,Y 517.943,Z 715.846,A -85,B 0,C 180,E1 -1372.472,E2 -1372.472} C_VEL
LIN {X 0,Y 518.4,Z 697.188,A -85,B 0,C 180,E1 -1373.074,E2 -1373.074} C_VEL
LIN {X 0,Y 518.685,Z 677.925,A -85,B 0,C 180,E1 -1373.474,E2 -1373.474} C_VEL
LIN {X 0,Y 520.261,Z 484.814,A -85,B 0,C 180,E1 -1376.297,E2 -1376.297} C_VEL
LIN {X 0,Y 519.249,Z 478.018,A -85,B 0,C 180,E1 -1376.479,E2 -1376.479} C_VEL
LIN {X 0,Y 520.255,Z 434.786,A -85,B 0,C 180,E1 -1379.599,E2 -1379.599} C_VEL
LIN {X 0,Y 521.689,Z 391.93,A -85,B 0,C 180,E1 -1382.847,E2 -1382.847} C_VEL
LIN {X 0,Y 520.188,Z 386.818,A -85,B 0,C 180,E1 -1383.349,E2 -1383.349} C_VEL
LIN {X 0,Y 512.619,Z 366.877,A -85,B 0,C 180,E1 -1385.401,E2 -1385.401} C_VEL
LIN {X 0,Y 512.617,Z 366.882,A -85,B 0,C 180,E1 -1388.721,E2 -1388.721} C_VEL
LIN {X 0,Y 512.589,Z 366.882,A -85,B 0,C 180,E1 -1392.163,E2 -1392.163} C_VEL
LIN {X 0,Y 512.638,Z 366.877,A -85,B 0,C 180,E1 -1395.557,E2 -1395.557} C_VEL
LIN {X 0,Y 512.603,Z 366.878,A -85,B 0,C 180,E1 -1398.903,E2 -1398.903} C_VEL
LIN {X 0,Y 512.644,Z 366.977,A -85,B 0,C 180,E1 -1401.839,E2 -1401.839} C_VEL
LIN {X 0,Y 515.331,Z 373.833,A -85,B 0,C 180,E1 -1402.702,E2 -1402.702} C_VEL
LIN {X 0,Y 523.255,Z 393.846,A -85,B 0,C 180,E1 -1405.156,E2 -1405.156} C_VEL
LIN {X 0,Y 523.629,Z 395.335,A -85,B 0,C 180,E1 -1405.317,E2 -1405.317} C_VEL
LIN {X 0,Y 521.974,Z 434.26,A -85,B 0,C 180,E1 -1408.534,E2 -1408.534} C_VEL
LIN {X 0,Y 520.235,Z 475.055,A -85,B 0,C 180,E1 -1411.846,E2 -1411.846} C_VEL
LIN {X 0,Y 518.478,Z 520.089,A -85,B 0,C 180,E1 -1415.444,E2 -1415.444} C_VEL
LIN {X 0,Y 516.855,Z 566.346,A -85,B 0,C 180,E1 -1419.089,E2 -1419.089} C_VEL
LIN {X 0,Y 516.136,Z 592.466,A -85,B 0,C 180,E1 -1421.1,E2 -1421.1} C_VEL
LIN {X 0,Y 516.75,Z 600.548,A -85,B 0,C 180,E1 -1421.263,E2 -1421.263} C_VEL
LIN {X 0,Y 516.068,Z 667.239,A -85,B 0,C 180,E1 -1422.272,E2 -1422.272} C_VEL
LIN {X 0,Y 515.413,Z 736.456,A -85,B 0,C 180,E1 -1423.358,E2 -1423.358} C_VEL
LIN {X 0,Y 515.166,Z 752.734,A -85,B 0,C 180,E1 -1423.828,E2 -1423.828} C_VEL
LIN {X 0,Y 514.833,Z 767.461,A -85,B 0,C 180,E1 -1424.454,E2 -1424.454} C_VEL
LIN {X 0,Y 514.392,Z 782.419,A -85,B 0,C 180,E1 -1425.305,E2 -1425.305} C_VEL
LIN {X 0,Y 513.912,Z 796.197,A -85,B 0,C 180,E1 -1426.326,E2 -1426.326} C_VEL
LIN {X 0,Y 513.473,Z 808.426,A -85,B 0,C 180,E1 -1427.46,E2 -1427.46} C_VEL
LIN {X 0,Y 513.019,Z 820.59,A -85,B 0,C 180,E1 -1428.875,E2 -1428.875} C_VEL
LIN {X 0,Y 512.69,Z 829.907,A -85,B 0,C 180,E1 -1430.231,E2 -1430.231} C_VEL
LIN {X 0,Y 512.419,Z 838.641,A -85,B 0,C 180,E1 -1431.811,E2 -1431.811} C_VEL
LIN {X 0,Y 512.223,Z 845.755,A -85,B 0,C 180,E1 -1433.502,E2 -1433.502} C_VEL
LIN {X 0,Y 512.122,Z 850.723,A -85,B 0,C 180,E1 -1435.072,E2 -1435.072} C_VEL
LIN {X 0,Y 512.063,Z 854.685,A -85,B 0,C 180,E1 -1436.866,E2 -1436.866} C_VEL
LIN {X 0,Y 512.05,Z 856.782,A -85,B 0,C 180,E1 -1438.657,E2 -1438.657} C_VEL
LIN {X 0,Y 512.054,Z 857.328,A -85,B 0,C 180,E1 -1440.335,E2 -1440.335} C_VEL
LIN {X 0,Y 512.075,Z 856.215,A -85,B 0,C 180,E1 -1442.238,E2 -1442.238} C_VEL
LIN {X 0,Y 512.124,Z 853.376,A -85,B 0,C 180,E1 -1444.03,E2 -1444.03} C_VEL
LIN {X 0,Y 512.235,Z 848.862,A -85,B 0,C 180,E1 -1445.825,E2 -1445.825} C_VEL
LIN {X 0,Y 512.429,Z 842.718,A -85,B 0,C 180,E1 -1447.512,E2 -1447.512} C_VEL
LIN {X 0,Y 512.691,Z 835.257,A -85,B 0,C 180,E1 -1449.089,E2 -1449.089} C_VEL
LIN {X 0,Y 513.028,Z 826.475,A -85,B 0,C 180,E1 -1450.556,E2 -1450.556} C_VEL
LIN {X 0,Y 513.448,Z 816.243,A -85,B 0,C 180,E1 -1451.912,E2 -1451.912} C_VEL
LIN {X 0,Y 513.931,Z 804.677,A -85,B 0,C 180,E1 -1453.157,E2 -1453.157} C_VEL
LIN {X 0,Y 514.403,Z 792.194,A -85,B 0,C 180,E1 -1454.234,E2 -1454.234} C_VEL
LIN {X 0,Y 514.876,Z 777.897,A -85,B 0,C 180,E1 -1455.198,E2 -1455.198} C_VEL
LIN {X 0,Y 515.276,Z 762.963,A -85,B 0,C 180,E1 -1455.965,E2 -1455.965} C_VEL
LIN {X 0,Y 515.532,Z 746.88,A -85,B 0,C 180,E1 -1456.546,E2 -1456.546} C_VEL
LIN {X 0,Y 515.686,Z 730.865,A -85,B 0,C 180,E1 -1456.913,E2 -1456.913} C_VEL
LIN {X 0,Y 517.38,Z 635.191,A -85,B 0,C 180,E1 -1458.558,E2 -1458.558} C_VEL
LIN {X 0,Y 518.395,Z 599.562,A -85,B 0,C 180,E1 -1459.228,E2 -1459.228} C_VEL
LIN {X 0,Y 519.028,Z 594.357,A -85,B 0,C 180,E1 -1459.637,E2 -1459.637} C_VEL
LIN {X 0,Y 522.255,Z 550.254,A -85,B 0,C 180,E1 -1463.407,E2 -1463.407} C_VEL
LIN {X 0,Y 526.313,Z 509.472,A -85,B 0,C 180,E1 -1467.064,E2 -1467.064} C_VEL
LIN {X 0,Y 531.03,Z 476.262,A -85,B 0,C 180,E1 -1470.204,E2 -1470.204} C_VEL
LIN {X 0,Y 536.554,Z 449.078,A -85,B 0,C 180,E1 -1472.965,E2 -1472.965} C_VEL
LIN {X 0,Y 542.201,Z 430.331,A -85,B 0,C 180,E1 -1475.038,E2 -1475.038} C_VEL
LIN {X 0,Y 545.77,Z 421.655,A -85,B 0,C 180,E1 -1476.106,E2 -1476.106} C_VEL
LIN {X 0,Y 545.656,Z 421.294,A -85,B 0,C 180,E1 -1476.445,E2 -1476.445} C_VEL
LIN {X 0,Y 538.789,Z 432.698,A -85,B 0,C 180,E1 -1477.588,E2 -1477.588} C_VEL
LIN {X 0,Y 533.567,Z 445.424,A -85,B 0,C 180,E1 -1478.78,E2 -1478.78} C_VEL
LIN {X 0,Y 530.423,Z 458.759,A -85,B 0,C 180,E1 -1480,E2 -1480} C_VEL
LIN {X 0,Y 529.456,Z 471.396,A -85,B 0,C 180,E1 -1481.157,E2 -1481.157} C_VEL
LIN {X 0,Y 530.483,Z 483.416,A -85,B 0,C 180,E1 -1482.289,E2 -1482.289} C_VEL
LIN {X 0,Y 533.446,Z 494.605,A -85,B 0,C 180,E1 -1483.388,E2 -1483.388} C_VEL
LIN {X 0,Y 537.809,Z 503.861,A -85,B 0,C 180,E1 -1484.349,E2 -1484.349} C_VEL
LIN {X 0,Y 544.135,Z 512.73,A -85,B 0,C 180,E1 -1485.326,E2 -1485.326} C_VEL
LIN {X 0,Y 551.512,Z 520.024,A -85,B 0,C 180,E1 -1486.182,E2 -1486.182} C_VEL
LIN {X 0,Y 560.427,Z 526.37,A -85,B 0,C 180,E1 -1487.01,E2 -1487.01} C_VEL
LIN {X 0,Y 569.854,Z 531.065,A -85,B 0,C 180,E1 -1487.768,E2 -1487.768} C_VEL
LIN {X 0,Y 574.556,Z 532.356,A -85,B 0,C 180,E1 -1488.293,E2 -1488.293} C_VEL
LIN {X 0,Y 577.752,Z 532.423,A -85,B 0,C 180,E1 -1488.834,E2 -1488.834} C_VEL
LIN {X 0,Y 579.885,Z 531.437,A -85,B 0,C 180,E1 -1489.455,E2 -1489.455} C_VEL
LIN {X 0,Y 580.543,Z 529.447,A -85,B 0,C 180,E1 -1490.086,E2 -1490.086} C_VEL
LIN {X 0,Y 579.632,Z 526.526,A -85,B 0,C 180,E1 -1490.691,E2 -1490.691} C_VEL
LIN {X 0,Y 577.132,Z 522.905,A -85,B 0,C 180,E1 -1491.224,E2 -1491.224} C_VEL
LIN {X 0,Y 570.368,Z 514.315,A -85,B 0,C 180,E1 -1492.089,E2 -1492.089} C_VEL
LIN {X 0,Y 569.925,Z 513.933,A -85,B 0,C 180,E1 -1492.146,E2 -1492.146} C_VEL
LIN {X 0,Y 565.79,Z 551.166,A -85,B 0,C 180,E1 -1492.688,E2 -1492.688} C_VEL
LIN {X 0,Y 562.669,Z 571.464,A -85,B 0,C 180,E1 -1493.101,E2 -1493.101} C_VEL
LIN {X 0,Y 560.386,Z 581.559,A -85,B 0,C 180,E1 -1493.4,E2 -1493.4} C_VEL
LIN {X 0,Y 557.168,Z 604.126,A -85,B 0,C 180,E1 -1493.568,E2 -1493.568} C_VEL
LIN {X 0,Y 551.828,Z 627.403,A -85,B 0,C 180,E1 -1493.726,E2 -1493.726} C_VEL
LIN {X 0,Y 545.704,Z 647.794,A -85,B 0,C 180,E1 -1493.974,E2 -1493.974} C_VEL
LIN {X 0,Y 540.954,Z 662.79,A -85,B 0,C 180,E1 -1494.327,E2 -1494.327} C_VEL
LIN {X 0,Y 538.428,Z 671.601,A -85,B 0,C 180,E1 -1494.658,E2 -1494.658} C_VEL
LIN {X 0,Y 533.693,Z 685.355,A -85,B 0,C 180,E1 -1494.955,E2 -1494.955} C_VEL
LIN {X 0,Y 530.356,Z 696.576,A -85,B 0,C 180,E1 -1495.36,E2 -1495.36} C_VEL
LIN {X 0,Y 528.778,Z 702.06,A -85,B 0,C 180,E1 -1495.571,E2 -1495.571} C_VEL
LIN {X 0,Y 525.733,Z 713.815,A -85,B 0,C 180,E1 -1496.036,E2 -1496.036} C_VEL
LIN {X 0,Y 525.008,Z 762.714,A -85,B 0,C 180,E1 -1496.814,E2 -1496.814} C_VEL
LIN {X 0,Y 524.25,Z 784.479,A -85,B 0,C 180,E1 -1497.354,E2 -1497.354} C_VEL
LIN {X 0,Y 523.313,Z 806.293,A -85,B 0,C 180,E1 -1498.11,E2 -1498.11} C_VEL
LIN {X 0,Y 522.177,Z 827.369,A -85,B 0,C 180,E1 -1499.052,E2 -1499.052} C_VEL
LIN {X 0,Y 520.914,Z 847.8,A -85,B 0,C 180,E1 -1500.189,E2 -1500.189} C_VEL
LIN {X 0,Y 519.539,Z 867.992,A -85,B 0,C 180,E1 -1501.555,E2 -1501.555} C_VEL
LIN {X 0,Y 518.136,Z 887.809,A -85,B 0,C 180,E1 -1503.156,E2 -1503.156} C_VEL
LIN {X 0,Y 516.837,Z 905.851,A -85,B 0,C 180,E1 -1504.874,E2 -1504.874} C_VEL
LIN {X 0,Y 515.591,Z 923.219,A -85,B 0,C 180,E1 -1506.817,E2 -1506.817} C_VEL
LIN {X 0,Y 514.513,Z 939.284,A -85,B 0,C 180,E1 -1508.929,E2 -1508.929} C_VEL
LIN {X 0,Y 513.638,Z 953.605,A -85,B 0,C 180,E1 -1511.147,E2 -1511.147} C_VEL
LIN {X 0,Y 512.963,Z 966.28,A -85,B 0,C 180,E1 -1513.466,E2 -1513.466} C_VEL
LIN {X 0,Y 512.485,Z 977.326,A -85,B 0,C 180,E1 -1515.884,E2 -1515.884} C_VEL
LIN {X 0,Y 512.189,Z 986.308,A -85,B 0,C 180,E1 -1518.286,E2 -1518.286} C_VEL
LIN {X 0,Y 512.024,Z 993.406,A -85,B 0,C 180,E1 -1520.672,E2 -1520.672} C_VEL
LIN {X 0,Y 511.948,Z 999.011,A -85,B 0,C 180,E1 -1523.157,E2 -1523.157} C_VEL
LIN {X 0,Y 511.92,Z 1002.876,A -85,B 0,C 180,E1 -1525.631,E2 -1525.631} C_VEL
LIN {X 0,Y 511.906,Z 1004.972,A -85,B 0,C 180,E1 -1528.097,E2 -1528.097} C_VEL
LIN {X 0,Y 511.893,Z 1005.406,A -85,B 0,C 180,E1 -1530.671,E2 -1530.671} C_VEL
LIN {X 0,Y 511.902,Z 1004.135,A -85,B 0,C 180,E1 -1533.135,E2 -1533.135} C_VEL
LIN {X 0,Y 511.92,Z 1001.336,A -85,B 0,C 180,E1 -1535.492,E2 -1535.492} C_VEL
LIN {X 0,Y 511.98,Z 996.692,A -85,B 0,C 180,E1 -1537.97,E2 -1537.97} C_VEL
LIN {X 0,Y 512.104,Z 990.266,A -85,B 0,C 180,E1 -1540.461,E2 -1540.461} C_VEL
LIN {X 0,Y 512.325,Z 982.27,A -85,B 0,C 180,E1 -1542.855,E2 -1542.855} C_VEL
LIN {X 0,Y 512.677,Z 972.844,A -85,B 0,C 180,E1 -1545.149,E2 -1545.149} C_VEL
LIN {X 0,Y 513.216,Z 961.49,A -85,B 0,C 180,E1 -1547.459,E2 -1547.459} C_VEL
LIN {X 0,Y 513.941,Z 948.569,A -85,B 0,C 180,E1 -1549.677,E2 -1549.677} C_VEL
LIN {X 0,Y 514.908,Z 933.356,A -85,B 0,C 180,E1 -1551.89,E2 -1551.89} C_VEL
LIN {X 0,Y 516.056,Z 916.707,A -85,B 0,C 180,E1 -1553.948,E2 -1553.948} C_VEL
LIN {X 0,Y 517.372,Z 898.477,A -85,B 0,C 180,E1 -1555.862,E2 -1555.862} C_VEL
LIN {X 0,Y 518.708,Z 879.604,A -85,B 0,C 180,E1 -1557.54,E2 -1557.54} C_VEL
LIN {X 0,Y 520.13,Z 859.623,A -85,B 0,C 180,E1 -1559.04,E2 -1559.04} C_VEL
LIN {X 0,Y 521.42,Z 839.754,A -85,B 0,C 180,E1 -1560.286,E2 -1560.286} C_VEL
LIN {X 0,Y 522.659,Z 818.907,A -85,B 0,C 180,E1 -1561.355,E2 -1561.355} C_VEL
LIN {X 0,Y 523.748,Z 797.073,A -85,B 0,C 180,E1 -1562.236,E2 -1562.236} C_VEL
LIN {X 0,Y 524.601,Z 775.371,A -85,B 0,C 180,E1 -1562.897,E2 -1562.897} C_VEL
LIN {X 0,Y 525.229,Z 752.626,A -85,B 0,C 180,E1 -1563.369,E2 -1563.369} C_VEL
LIN {X 0,Y 525.811,Z 712.791,A -85,B 0,C 180,E1 -1563.99,E2 -1563.99} C_VEL
LIN {X 0,Y 528.774,Z 702.072,A -85,B 0,C 180,E1 -1564.428,E2 -1564.428} C_VEL
LIN {X 0,Y 530.353,Z 696.588,A -85,B 0,C 180,E1 -1564.639,E2 -1564.639} C_VEL
LIN {X 0,Y 533.692,Z 685.36,A -85,B 0,C 180,E1 -1565.045,E2 -1565.045} C_VEL
LIN {X 0,Y 538.784,Z 670.425,A -85,B 0,C 180,E1 -1565.38,E2 -1565.38} C_VEL
LIN {X 0,Y 541.702,Z 660.357,A -85,B 0,C 180,E1 -1565.745,E2 -1565.745} C_VEL
LIN {X 0,Y 546.851,Z 644.181,A -85,B 0,C 180,E1 -1566.085,E2 -1566.085} C_VEL
LIN {X 0,Y 552.989,Z 623.013,A -85,B 0,C 180,E1 -1566.307,E2 -1566.307} C_VEL
LIN {X 0,Y 557.934,Z 599.812,A -85,B 0,C 180,E1 -1566.462,E2 -1566.462} C_VEL
LIN {X 0,Y 560.685,Z 579.821,A -85,B 0,C 180,E1 -1566.636,E2 -1566.636} C_VEL
LIN {X 0,Y 563.149,Z 568.936,A -85,B 0,C 180,E1 -1566.961,E2 -1566.961} C_VEL
LIN {X 0,Y 566.546,Z 545.185,A -85,B 0,C 180,E1 -1567.412,E2 -1567.412} C_VEL
LIN {X 0,Y 570.056,Z 513.862,A -85,B 0,C 180,E1 -1567.871,E2 -1567.871} C_VEL
LIN {X 0,Y 576.849,Z 522.568,A -85,B 0,C 180,E1 -1568.735,E2 -1568.735} C_VEL
LIN {X 0,Y 579.47,Z 526.228,A -85,B 0,C 180,E1 -1569.258,E2 -1569.258} C_VEL
LIN {X 0,Y 580.521,Z 529.164,A -85,B 0,C 180,E1 -1569.845,E2 -1569.845} C_VEL
LIN {X 0,Y 580.189,Z 531.037,A -85,B 0,C 180,E1 -1570.389,E2 -1570.389} C_VEL
LIN {X 0,Y 578.616,Z 532.213,A -85,B 0,C 180,E1 -1570.963,E2 -1570.963} C_VEL
LIN {X 0,Y 575.71,Z 532.495,A -85,B 0,C 180,E1 -1571.537,E2 -1571.537} C_VEL
LIN {X 0,Y 571.5,Z 531.631,A -85,B 0,C 180,E1 -1572.072,E2 -1572.072} C_VEL
LIN {X 0,Y 562.311,Z 527.711,A -85,B 0,C 180,E1 -1573.046,E2 -1573.046} C_VEL
LIN {X 0,Y 554.046,Z 522.135,A -85,B 0,C 180,E1 -1574.09,E2 -1574.09} C_VEL
LIN {X 0,Y 547.101,Z 515.073,A -85,B 0,C 180,E1 -1575.161,E2 -1575.161} C_VEL
LIN {X 0,Y 541.719,Z 506.945,A -85,B 0,C 180,E1 -1576.2,E2 -1576.2} C_VEL
LIN {X 0,Y 537.441,Z 496.995,A -85,B 0,C 180,E1 -1577.295,E2 -1577.295} C_VEL
LIN {X 0,Y 534.674,Z 485.338,A -85,B 0,C 180,E1 -1578.418,E2 -1578.418} C_VEL
LIN {X 0,Y 533.296,Z 471.058,A -85,B 0,C 180,E1 -1579.627,E2 -1579.627} C_VEL
LIN {X 0,Y 533.609,Z 452.749,A -85,B 0,C 180,E1 -1580.981,E2 -1580.981} C_VEL
LIN {X 0,Y 536.279,Z 411.573,A -85,B 0,C 180,E1 -1583.903,E2 -1583.903} C_VEL
LIN {X 0,Y 536.314,Z 409.843,A -85,B 0,C 180,E1 -1584.038,E2 -1584.038} C_VEL
LIN {X 0,Y 525.948,Z 391.02,A -85,B 0,C 180,E1 -1586.968,E2 -1586.968} C_VEL
LIN {X 0,Y 520.357,Z 381.19,A -85,B 0,C 180,E1 -1588.62,E2 -1588.62} C_VEL
LIN {X 0,Y 517.581,Z 376.316,A -85,B 0,C 180,E1 -1589.466,E2 -1589.466} C_VEL
LIN {X 0,Y 515.592,Z 372.626,A -85,B 0,C 180,E1 -1590.107,E2 -1590.107} C_VEL
LIN {X 0,Y 513.086,Z 368.724,A -85,B 0,C 180,E1 -1590.845,E2 -1590.845} C_VEL
LIN {X 0,Y 512.612,Z 366.881,A -85,B 0,C 180,E1 -1591.137,E2 -1591.137} C_VEL
LIN {X 0,Y 512.618,Z 366.881,A -85,B 0,C 180,E1 -1594.713,E2 -1594.713} C_VEL
LIN {X 0,Y 512.645,Z 366.877,A -85,B 0,C 180,E1 -1598.184,E2 -1598.184} C_VEL
LIN {X 0,Y 512.631,Z 366.881,A -85,B 0,C 180,E1 -1601.816,E2 -1601.816} C_VEL
LIN {X 0,Y 512.641,Z 366.881,A -85,B 0,C 180,E1 -1605.312,E2 -1605.312} C_VEL
LIN {X 0,Y 512.629,Z 366.882,A -85,B 0,C 180,E1 -1608.835,E2 -1608.835} C_VEL
LIN {X 0,Y 512.632,Z 366.879,A -85,B 0,C 180,E1 -1612.266,E2 -1612.266} C_VEL
LIN {X 0,Y 512.598,Z 366.884,A -85,B 0,C 180,E1 -1615.862,E2 -1615.862} C_VEL
LIN {X 0,Y 512.642,Z 366.88,A -85,B 0,C 180,E1 -1619.33,E2 -1619.33} C_VEL
LIN {X 0,Y 512.612,Z 366.885,A -85,B 0,C 180,E1 -1622.683,E2 -1622.683} C_VEL
LIN {X 0,Y 512.641,Z 366.882,A -85,B 0,C 180,E1 -1626.158,E2 -1626.158} C_VEL
LIN {X 0,Y 512.643,Z 366.882,A -85,B 0,C 180,E1 -1629.543,E2 -1629.543} C_VEL
LIN {X 0,Y 512.647,Z 366.879,A -85,B 0,C 180,E1 -1633.076,E2 -1633.076} C_VEL
LIN {X 0,Y 512.609,Z 366.882,A -85,B 0,C 180,E1 -1636.546,E2 -1636.546} C_VEL
LIN {X 0,Y 512.625,Z 366.879,A -85,B 0,C 180,E1 -1640.077,E2 -1640.077} C_VEL
LIN {X 0,Y 512.627,Z 366.878,A -85,B 0,C 180,E1 -1643.447,E2 -1643.447} C_VEL
LIN {X 0,Y 512.612,Z 366.879,A -85,B 0,C 180,E1 -1646.952,E2 -1646.952} C_VEL
LIN {X 0,Y 512.648,Z 366.878,A -85,B 0,C 180,E1 -1650.471,E2 -1650.471} C_VEL
LIN {X 0,Y 512.646,Z 366.876,A -85,B 0,C 180,E1 -1654.04,E2 -1654.04} C_VEL
LIN {X 0,Y 512.63,Z 366.867,A -85,B 0,C 180,E1 -1657.484,E2 -1657.484} C_VEL
LIN {X 0,Y 512.6,Z 366.877,A -85,B 0,C 180,E1 -1660.95,E2 -1660.95} C_VEL
LIN {X 0,Y 512.644,Z 366.879,A -85,B 0,C 180,E1 -1664.292,E2 -1664.292} C_VEL
LIN {X 0,Y 512.62,Z 366.878,A -85,B 0,C 180,E1 -1665.967,E2 -1665.967} C_VEL
LIN {X 0,Y 511.631,Z 367.005,A -85,B 0,C 180,E1 -1666.828,E2 -1666.828} C_VEL
LIN {X 0,Y 505.188,Z 367.818,A -85,B 0,C 180,E1 -1669.248,E2 -1669.248} C_VEL
LIN {X 0,Y 504.687,Z 367.871,A -85,B 0,C 180,E1 -1669.879,E2 -1669.879} C_VEL
LIN {X 0,Y 504.703,Z 367.87,A -85,B 0,C 180,E1 -1673.395,E2 -1673.395} C_VEL
LIN {X 0,Y 504.681,Z 367.959,A -85,B 0,C 180,E1 -1674.174,E2 -1674.174} C_VEL
LIN {X 0,Y 513.904,Z 391.922,A -85,B 0,C 180,E1 -1676.683,E2 -1676.683} C_VEL
LIN {X 0,Y 514.601,Z 394.959,A -85,B 0,C 180,E1 -1676.975,E2 -1676.975} C_VEL
LIN {X 0,Y 513.001,Z 438.92,A -85,B 0,C 180,E1 -1680.327,E2 -1680.327} C_VEL
LIN {X 0,Y 512.115,Z 478.289,A -85,B 0,C 180,E1 -1683.158,E2 -1683.158} C_VEL
LIN {X 0,Y 512.332,Z 480.799,A -85,B 0,C 180,E1 -1683.273,E2 -1683.273} C_VEL
LIN {X 0,Y 513.283,Z 488.704,A -85,B 0,C 180,E1 -1683.451,E2 -1683.451} C_VEL
LIN {X 0,Y 511.283,Z 687.571,A -85,B 0,C 180,E1 -1686.418,E2 -1686.418} C_VEL
LIN {X 0,Y 510.934,Z 705.896,A -85,B 0,C 180,E1 -1686.891,E2 -1686.891} C_VEL
LIN {X 0,Y 510.4,Z 723.375,A -85,B 0,C 180,E1 -1687.543,E2 -1687.543} C_VEL
LIN {X 0,Y 509.67,Z 740.999,A -85,B 0,C 180,E1 -1688.417,E2 -1688.417} C_VEL
LIN {X 0,Y 508.849,Z 757.578,A -85,B 0,C 180,E1 -1689.468,E2 -1689.468} C_VEL
LIN {X 0,Y 508.009,Z 773.153,A -85,B 0,C 180,E1 -1690.692,E2 -1690.692} C_VEL
LIN {X 0,Y 507.124,Z 787.733,A -85,B 0,C 180,E1 -1692.087,E2 -1692.087} C_VEL
LIN {X 0,Y 506.315,Z 800.79,A -85,B 0,C 180,E1 -1693.597,E2 -1693.597} C_VEL
LIN {X 0,Y 505.544,Z 813.22,A -85,B 0,C 180,E1 -1695.336,E2 -1695.336} C_VEL
LIN {X 0,Y 504.932,Z 824.069,A -85,B 0,C 180,E1 -1697.187,E2 -1697.187} C_VEL
LIN {X 0,Y 504.483,Z 833.391,A -85,B 0,C 180,E1 -1699.148,E2 -1699.148} C_VEL
LIN {X 0,Y 504.161,Z 841.179,A -85,B 0,C 180,E1 -1701.216,E2 -1701.216} C_VEL
LIN {X 0,Y 503.991,Z 847.378,A -85,B 0,C 180,E1 -1703.393,E2 -1703.393} C_VEL
LIN {X 0,Y 503.928,Z 851.707,A -85,B 0,C 180,E1 -1705.562,E2 -1705.562} C_VEL
LIN {X 0,Y 503.911,Z 854.358,A -85,B 0,C 180,E1 -1707.612,E2 -1707.612} C_VEL
LIN {X 0,Y 503.909,Z 855.43,A -85,B 0,C 180,E1 -1709.659,E2 -1709.659} C_VEL
LIN {X 0,Y 503.913,Z 854.874,A -85,B 0,C 180,E1 -1711.82,E2 -1711.82} C_VEL
LIN {X 0,Y 503.92,Z 852.724,A -85,B 0,C 180,E1 -1713.869,E2 -1713.869} C_VEL
LIN {X 0,Y 503.966,Z 848.653,A -85,B 0,C 180,E1 -1716.151,E2 -1716.151} C_VEL
LIN {X 0,Y 504.106,Z 842.968,A -85,B 0,C 180,E1 -1718.325,E2 -1718.325} C_VEL
LIN {X 0,Y 504.382,Z 835.69,A -85,B 0,C 180,E1 -1720.393,E2 -1720.393} C_VEL
LIN {X 0,Y 504.796,Z 826.911,A -85,B 0,C 180,E1 -1722.352,E2 -1722.352} C_VEL
LIN {X 0,Y 505.339,Z 816.675,A -85,B 0,C 180,E1 -1724.203,E2 -1724.203} C_VEL
LIN {X 0,Y 506.048,Z 804.963,A -85,B 0,C 180,E1 -1725.941,E2 -1725.941} C_VEL
LIN {X 0,Y 506.86,Z 791.696,A -85,B 0,C 180,E1 -1727.567,E2 -1727.567} C_VEL
LIN {X 0,Y 507.779,Z 776.694,A -85,B 0,C 180,E1 -1729.079,E2 -1729.079} C_VEL
LIN {X 0,Y 508.661,Z 761.146,A -85,B 0,C 180,E1 -1730.361,E2 -1730.361} C_VEL
LIN {X 0,Y 509.456,Z 745.478,A -85,B 0,C 180,E1 -1731.411,E2 -1731.411} C_VEL
LIN {X 0,Y 510.181,Z 729.13,A -85,B 0,C 180,E1 -1732.286,E2 -1732.286} C_VEL
LIN {X 0,Y 510.786,Z 711.127,A -85,B 0,C 180,E1 -1733.025,E2 -1733.025} C_VEL
LIN {X 0,Y 511.212,Z 692.818,A -85,B 0,C 180,E1 -1733.558,E2 -1733.558} C_VEL
LIN {X 0,Y 511.458,Z 671.318,A -85,B 0,C 180,E1 -1733.942,E2 -1733.942} C_VEL
LIN {X 0,Y 513.134,Z 485.859,A -85,B 0,C 180,E1 -1736.692,E2 -1736.692} C_VEL
LIN {X 0,Y 512.123,Z 479.215,A -85,B 0,C 180,E1 -1736.871,E2 -1736.871} C_VEL
LIN {X 0,Y 512.875,Z 442.572,A -85,B 0,C 180,E1 -1739.489,E2 -1739.489} C_VEL
LIN {X 0,Y 514.529,Z 397.659,A -85,B 0,C 180,E1 -1742.914,E2 -1742.914} C_VEL
LIN {X 0,Y 514.442,Z 393.626,A -85,B 0,C 180,E1 -1743.236,E2 -1743.236} C_VEL
LIN {X 0,Y 506.962,Z 373.948,A -85,B 0,C 180,E1 -1745.301,E2 -1745.301} C_VEL
LIN {X 0,Y 504.652,Z 367.874,A -85,B 0,C 180,E1 -1745.942,E2 -1745.942} C_VEL
LIN {X 0,Y 504.701,Z 367.867,A -85,B 0,C 180,E1 -1749.343,E2 -1749.343} C_VEL
LIN {X 0,Y 504.665,Z 367.873,A -85,B 0,C 180,E1 -1752.689,E2 -1752.689} C_VEL
LIN {X 0,Y 504.653,Z 367.873,A -85,B 0,C 180,E1 -1756.153,E2 -1756.153} C_VEL
LIN {X 0,Y 504.709,Z 367.869,A -85,B 0,C 180,E1 -1759.623,E2 -1759.623} C_VEL
LIN {X 0,Y 504.681,Z 367.875,A -85,B 0,C 180,E1 -1761.168,E2 -1761.168} C_VEL
LIN {X 0,Y 514.405,Z 391.967,A -85,B 0,C 180,E1 -1764.244,E2 -1764.244} C_VEL
LIN {X 0,Y 516.723,Z 398.418,A -85,B 0,C 180,E1 -1765.01,E2 -1765.01} C_VEL
LIN {X 0,Y 514.901,Z 437.463,A -85,B 0,C 180,E1 -1768.27,E2 -1768.27} C_VEL
LIN {X 0,Y 513.004,Z 478.948,A -85,B 0,C 180,E1 -1771.667,E2 -1771.667} C_VEL
LIN {X 0,Y 511.148,Z 523.435,A -85,B 0,C 180,E1 -1775.253,E2 -1775.253} C_VEL
LIN {X 0,Y 509.43,Z 569.158,A -85,B 0,C 180,E1 -1778.89,E2 -1778.89} C_VEL
LIN {X 0,Y 508.719,Z 593.258,A -85,B 0,C 180,E1 -1780.762,E2 -1780.762} C_VEL
LIN {X 0,Y 509.36,Z 601.219,A -85,B 0,C 180,E1 -1780.927,E2 -1780.927} C_VEL
LIN {X 0,Y 507.807,Z 737.149,A -85,B 0,C 180,E1 -1783.09,E2 -1783.09} C_VEL
LIN {X 0,Y 507.545,Z 753.844,A -85,B 0,C 180,E1 -1783.579,E2 -1783.579} C_VEL
LIN {X 0,Y 507.197,Z 768.558,A -85,B 0,C 180,E1 -1784.214,E2 -1784.214} C_VEL
LIN {X 0,Y 506.696,Z 784.332,A -85,B 0,C 180,E1 -1785.136,E2 -1785.136} C_VEL
LIN {X 0,Y 506.186,Z 797.953,A -85,B 0,C 180,E1 -1786.172,E2 -1786.172} C_VEL
LIN {X 0,Y 505.671,Z 811.136,A -85,B 0,C 180,E1 -1787.437,E2 -1787.437} C_VEL
LIN {X 0,Y 505.209,Z 822.545,A -85,B 0,C 180,E1 -1788.816,E2 -1788.816} C_VEL
LIN {X 0,Y 504.833,Z 832.448,A -85,B 0,C 180,E1 -1790.308,E2 -1790.308} C_VEL
LIN {X 0,Y 504.547,Z 840.898,A -85,B 0,C 180,E1 -1791.911,E2 -1791.911} C_VEL
LIN {X 0,Y 504.342,Z 847.773,A -85,B 0,C 180,E1 -1793.626,E2 -1793.626} C_VEL
LIN {X 0,Y 504.228,Z 852.897,A -85,B 0,C 180,E1 -1795.336,E2 -1795.336} C_VEL
LIN {X 0,Y 504.177,Z 856.652,A -85,B 0,C 180,E1 -1797.272,E2 -1797.272} C_VEL
LIN {X 0,Y 504.165,Z 858.438,A -85,B 0,C 180,E1 -1799.091,E2 -1799.091} C_VEL
LIN {X 0,Y 504.182,Z 858.54,A -85,B 0,C 180,E1 -1801.022,E2 -1801.022} C_VEL
LIN {X 0,Y 504.221,Z 856.9,A -85,B 0,C 180,E1 -1802.841,E2 -1802.841} C_VEL
LIN {X 0,Y 504.303,Z 853.643,A -85,B 0,C 180,E1 -1804.662,E2 -1804.662} C_VEL
LIN {X 0,Y 504.479,Z 848.487,A -85,B 0,C 180,E1 -1806.486,E2 -1806.486} C_VEL
LIN {X 0,Y 504.737,Z 841.814,A -85,B 0,C 180,E1 -1808.2,E2 -1808.2} C_VEL
LIN {X 0,Y 505.1,Z 832.98,A -85,B 0,C 180,E1 -1809.917,E2 -1809.917} C_VEL
LIN {X 0,Y 505.533,Z 823.206,A -85,B 0,C 180,E1 -1811.407,E2 -1811.407} C_VEL
LIN {X 0,Y 506.07,Z 811.326,A -85,B 0,C 180,E1 -1812.842,E2 -1812.842} C_VEL
LIN {X 0,Y 506.592,Z 799.431,A -85,B 0,C 180,E1 -1813.991,E2 -1813.991} C_VEL
LIN {X 0,Y 507.101,Z 785.903,A -85,B 0,C 180,E1 -1815.027,E2 -1815.027} C_VEL
LIN {X 0,Y 507.556,Z 771.41,A -85,B 0,C 180,E1 -1815.892,E2 -1815.892} C_VEL
LIN {X 0,Y 507.896,Z 755.393,A -85,B 0,C 180,E1 -1816.585,E2 -1816.585} C_VEL
LIN {X 0,Y 508.096,Z 739.548,A -85,B 0,C 180,E1 -1817.05,E2 -1817.05} C_VEL
LIN {X 0,Y 510.009,Z 643.779,A -85,B 0,C 180,E1 -1818.803,E2 -1818.803} C_VEL
LIN {X 0,Y 511.368,Z 602.209,A -85,B 0,C 180,E1 -1819.622,E2 -1819.622} C_VEL
LIN {X 0,Y 512.145,Z 598.837,A -85,B 0,C 180,E1 -1819.858,E2 -1819.858} C_VEL
LIN {X 0,Y 515.203,Z 559.567,A -85,B 0,C 180,E1 -1823.262,E2 -1823.262} C_VEL
LIN {X 0,Y 519.589,Z 518.169,A -85,B 0,C 180,E1 -1827.009,E2 -1827.009} C_VEL
LIN {X 0,Y 524.222,Z 486.815,A -85,B 0,C 180,E1 -1830.011,E2 -1830.011} C_VEL
LIN {X 0,Y 529.821,Z 460.166,A -85,B 0,C 180,E1 -1832.729,E2 -1832.729} C_VEL
LIN {X 0,Y 535.943,Z 440.268,A -85,B 0,C 180,E1 -1834.941,E2 -1834.941} C_VEL
LIN {X 0,Y 540.466,Z 429.845,A -85,B 0,C 180,E1 -1836.212,E2 -1836.212} C_VEL
LIN {X 0,Y 532.998,Z 441.851,A -85,B 0,C 180,E1 -1837.43,E2 -1837.43} C_VEL
LIN {X 0,Y 527.837,Z 453.888,A -85,B 0,C 180,E1 -1838.612,E2 -1838.612} C_VEL
LIN {X 0,Y 524.726,Z 466.413,A -85,B 0,C 180,E1 -1839.833,E2 -1839.833} C_VEL
LIN {X 0,Y 523.803,Z 478.89,A -85,B 0,C 180,E1 -1841.062,E2 -1841.062} C_VEL
LIN {X 0,Y 525.001,Z 490.618,A -85,B 0,C 180,E1 -1842.243,E2 -1842.243} C_VEL
LIN {X 0,Y 528.128,Z 501.338,A -85,B 0,C 180,E1 -1843.365,E2 -1843.365} C_VEL
LIN {X 0,Y 532.942,Z 510.875,A -85,B 0,C 180,E1 -1844.41,E2 -1844.41} C_VEL
LIN {X 0,Y 539.961,Z 520.045,A -85,B 0,C 180,E1 -1845.472,E2 -1845.472} C_VEL
LIN {X 0,Y 548.137,Z 527.567,A -85,B 0,C 180,E1 -1846.399,E2 -1846.399} C_VEL
LIN {X 0,Y 557.94,Z 534.057,A -85,B 0,C 180,E1 -1847.285,E2 -1847.285} C_VEL
LIN {X 0,Y 567.485,Z 538.492,A -85,B 0,C 180,E1 -1848.032,E2 -1848.032} C_VEL
LIN {X 0,Y 572.241,Z 539.687,A -85,B 0,C 180,E1 -1848.553,E2 -1848.553} C_VEL
LIN {X 0,Y 575.481,Z 539.693,A -85,B 0,C 180,E1 -1849.093,E2 -1849.093} C_VEL
LIN {X 0,Y 577.48,Z 538.836,A -85,B 0,C 180,E1 -1849.642,E2 -1849.642} C_VEL
LIN {X 0,Y 578.345,Z 536.881,A -85,B 0,C 180,E1 -1850.293,E2 -1850.293} C_VEL
LIN {X 0,Y 577.591,Z 534.049,A -85,B 0,C 180,E1 -1850.906,E2 -1850.906} C_VEL
LIN {X 0,Y 575.226,Z 530.521,A -85,B 0,C 180,E1 -1851.453,E2 -1851.453} C_VEL
LIN {X 0,Y 573.434,Z 528.571,A -85,B 0,C 180,E1 -1851.698,E2 -1851.698} C_VEL
LIN {X 0,Y 569.858,Z 554.522,A -85,B 0,C 180,E1 -1852.057,E2 -1852.057} C_VEL
LIN {X 0,Y 565.828,Z 573.886,A -85,B 0,C 180,E1 -1852.396,E2 -1852.396} C_VEL
LIN {X 0,Y 563.292,Z 583.818,A -85,B 0,C 180,E1 -1852.663,E2 -1852.663} C_VEL
LIN {X 0,Y 557.914,Z 606.101,A -85,B 0,C 180,E1 -1852.763,E2 -1852.763} C_VEL
LIN {X 0,Y 550.455,Z 628.689,A -85,B 0,C 180,E1 -1852.911,E2 -1852.911} C_VEL
LIN {X 0,Y 542.796,Z 648.556,A -85,B 0,C 180,E1 -1853.192,E2 -1853.192} C_VEL
LIN {X 0,Y 537.234,Z 663.602,A -85,B 0,C 180,E1 -1853.58,E2 -1853.58} C_VEL
LIN {X 0,Y 534.531,Z 672.411,A -85,B 0,C 180,E1 -1853.907,E2 -1853.907} C_VEL
LIN {X 0,Y 528.971,Z 686.261,A -85,B 0,C 180,E1 -1854.262,E2 -1854.262} C_VEL
LIN {X 0,Y 525.269,Z 698.057,A -85,B 0,C 180,E1 -1854.709,E2 -1854.709} C_VEL
LIN {X 0,Y 520.852,Z 712.93,A -85,B 0,C 180,E1 -1855.307,E2 -1855.307} C_VEL
LIN {X 0,Y 519.005,Z 721.141,A -85,B 0,C 180,E1 -1855.655,E2 -1855.655} C_VEL
LIN {X 0,Y 518.3,Z 763.054,A -85,B 0,C 180,E1 -1856.336,E2 -1856.336} C_VEL
LIN {X 0,Y 517.472,Z 784.97,A -85,B 0,C 180,E1 -1856.888,E2 -1856.888} C_VEL
LIN {X 0,Y 516.432,Z 807.05,A -85,B 0,C 180,E1 -1857.666,E2 -1857.666} C_VEL
LIN {X 0,Y 515.223,Z 827.651,A -85,B 0,C 180,E1 -1858.603,E2 -1858.603} C_VEL
LIN {X 0,Y 513.822,Z 848.292,A -85,B 0,C 180,E1 -1859.767,E2 -1859.767} C_VEL
LIN {X 0,Y 512.35,Z 868.115,A -85,B 0,C 180,E1 -1861.128,E2 -1861.128} C_VEL
LIN {X 0,Y 510.817,Z 887.806,A -85,B 0,C 180,E1 -1862.74,E2 -1862.74} C_VEL
LIN {X 0,Y 509.382,Z 905.836,A -85,B 0,C 180,E1 -1864.478,E2 -1864.478} C_VEL
LIN {X 0,Y 508.012,Z 923.219,A -85,B 0,C 180,E1 -1866.45,E2 -1866.45} C_VEL
LIN {X 0,Y 506.806,Z 939.472,A -85,B 0,C 180,E1 -1868.62,E2 -1868.62} C_VEL
LIN {X 0,Y 505.838,Z 953.809,A -85,B 0,C 180,E1 -1870.879,E2 -1870.879} C_VEL
LIN {X 0,Y 505.102,Z 966.283,A -85,B 0,C 180,E1 -1873.201,E2 -1873.201} C_VEL
LIN {X 0,Y 504.562,Z 977.329,A -85,B 0,C 180,E1 -1875.658,E2 -1875.658} C_VEL
LIN {X 0,Y 504.225,Z 986.307,A -85,B 0,C 180,E1 -1878.098,E2 -1878.098} C_VEL
LIN {X 0,Y 504.035,Z 993.406,A -85,B 0,C 180,E1 -1880.523,E2 -1880.523} C_VEL
LIN {X 0,Y 503.945,Z 998.805,A -85,B 0,C 180,E1 -1882.934,E2 -1882.934} C_VEL
LIN {X 0,Y 503.917,Z 1002.738,A -85,B 0,C 180,E1 -1885.447,E2 -1885.447} C_VEL
LIN {X 0,Y 503.91,Z 1004.907,A -85,B 0,C 180,E1 -1887.953,E2 -1887.953} C_VEL
LIN {X 0,Y 503.893,Z 1005.431,A -85,B 0,C 180,E1 -1890.568,E2 -1890.568} C_VEL
LIN {X 0,Y 503.897,Z 1004.328,A -85,B 0,C 180,E1 -1892.957,E2 -1892.957} C_VEL
LIN {X 0,Y 503.911,Z 1001.656,A -85,B 0,C 180,E1 -1895.351,E2 -1895.351} C_VEL
LIN {X 0,Y 503.975,Z 997.203,A -85,B 0,C 180,E1 -1897.868,E2 -1897.868} C_VEL
LIN {X 0,Y 504.103,Z 991.105,A -85,B 0,C 180,E1 -1900.333,E2 -1900.333} C_VEL
LIN {X 0,Y 504.347,Z 983.111,A -85,B 0,C 180,E1 -1902.828,E2 -1902.828} C_VEL
LIN {X 0,Y 504.749,Z 973.366,A -85,B 0,C 180,E1 -1905.275,E2 -1905.275} C_VEL
LIN {X 0,Y 505.341,Z 962.124,A -85,B 0,C 180,E1 -1907.621,E2 -1907.621} C_VEL
LIN {X 0,Y 506.18,Z 948.631,A -85,B 0,C 180,E1 -1909.982,E2 -1909.982} C_VEL
LIN {X 0,Y 507.249,Z 933.358,A -85,B 0,C 180,E1 -1912.238,E2 -1912.238} C_VEL
LIN {X 0,Y 508.523,Z 916.711,A -85,B 0,C 180,E1 -1914.325,E2 -1914.325} C_VEL
LIN {X 0,Y 509.956,Z 898.747,A -85,B 0,C 180,E1 -1916.24,E2 -1916.24} C_VEL
LIN {X 0,Y 511.392,Z 880.342,A -85,B 0,C 180,E1 -1917.904,E2 -1917.904} C_VEL
LIN {X 0,Y 512.927,Z 860.51,A -85,B 0,C 180,E1 -1919.421,E2 -1919.421} C_VEL
LIN {X 0,Y 514.336,Z 840.764,A -85,B 0,C 180,E1 -1920.683,E2 -1920.683} C_VEL
LIN {X 0,Y 515.682,Z 820.192,A -85,B 0,C 180,E1 -1921.763,E2 -1921.763} C_VEL
LIN {X 0,Y 516.88,Z 798.499,A -85,B 0,C 180,E1 -1922.663,E2 -1922.663} C_VEL
LIN {X 0,Y 517.811,Z 777.109,A -85,B 0,C 180,E1 -1923.335,E2 -1923.335} C_VEL
LIN {X 0,Y 518.5,Z 754.843,A -85,B 0,C 180,E1 -1923.819,E2 -1923.819} C_VEL
LIN {X 0,Y 519.034,Z 720.232,A -85,B 0,C 180,E1 -1924.362,E2 -1924.362} C_VEL
LIN {X 0,Y 523.233,Z 704.499,A -85,B 0,C 180,E1 -1925.046,E2 -1925.046} C_VEL
LIN {X 0,Y 525.538,Z 697.026,A -85,B 0,C 180,E1 -1925.336,E2 -1925.336} C_VEL
LIN {X 0,Y 529.374,Z 685.163,A -85,B 0,C 180,E1 -1925.772,E2 -1925.772} C_VEL
LIN {X 0,Y 534.945,Z 671.155,A -85,B 0,C 180,E1 -1926.135,E2 -1926.135} C_VEL
LIN {X 0,Y 538.413,Z 660.198,A -85,B 0,C 180,E1 -1926.525,E2 -1926.525} C_VEL
LIN {X 0,Y 544.619,Z 643.895,A -85,B 0,C 180,E1 -1926.894,E2 -1926.894} C_VEL
LIN {X 0,Y 552.466,Z 623.119,A -85,B 0,C 180,E1 -1927.135,E2 -1927.135} C_VEL
LIN {X 0,Y 559.461,Z 600.485,A -85,B 0,C 180,E1 -1927.264,E2 -1927.264} C_VEL
LIN {X 0,Y 563.707,Z 582.015,A -85,B 0,C 180,E1 -1927.369,E2 -1927.369} C_VEL
LIN {X 0,Y 566.789,Z 569.788,A -85,B 0,C 180,E1 -1927.692,E2 -1927.692} C_VEL
LIN {X 0,Y 571.07,Z 547.204,A -85,B 0,C 180,E1 -1928.046,E2 -1928.046} C_VEL
LIN {X 0,Y 573.45,Z 528.489,A -85,B 0,C 180,E1 -1928.305,E2 -1928.305} C_VEL
LIN {X 0,Y 576.633,Z 532.402,A -85,B 0,C 180,E1 -1928.816,E2 -1928.816} C_VEL
LIN {X 0,Y 578.17,Z 535.571,A -85,B 0,C 180,E1 -1929.395,E2 -1929.395} C_VEL
LIN {X 0,Y 578.162,Z 537.87,A -85,B 0,C 180,E1 -1929.994,E2 -1929.994} C_VEL
LIN {X 0,Y 576.756,Z 539.302,A -85,B 0,C 180,E1 -1930.597,E2 -1930.597} C_VEL
LIN {X 0,Y 573.965,Z 539.812,A -85,B 0,C 180,E1 -1931.188,E2 -1931.188} C_VEL
LIN {X 0,Y 570.326,Z 539.328,A -85,B 0,C 180,E1 -1931.683,E2 -1931.683} C_VEL
LIN {X 0,Y 560.509,Z 535.7,A -85,B 0,C 180,E1 -1932.698,E2 -1932.698} C_VEL
LIN {X 0,Y 552.005,Z 530.663,A -85,B 0,C 180,E1 -1933.721,E2 -1933.721} C_VEL
LIN {X 0,Y 544.273,Z 523.866,A -85,B 0,C 180,E1 -1934.838,E2 -1934.838} C_VEL
LIN {X 0,Y 537.676,Z 515.203,A -85,B 0,C 180,E1 -1936.026,E2 -1936.026} C_VEL
LIN {X 0,Y 532.649,Z 504.968,A -85,B 0,C 180,E1 -1937.219,E2 -1937.219} C_VEL
LIN {X 0,Y 529.427,Z 494.002,A -85,B 0,C 180,E1 -1938.335,E2 -1938.335} C_VEL
LIN {X 0,Y 527.506,Z 480.031,A -85,B 0,C 180,E1 -1939.591,E2 -1939.591} C_VEL
LIN {X 0,Y 527.187,Z 463.751,A -85,B 0,C 180,E1 -1940.869,E2 -1940.869} C_VEL
LIN {X 0,Y 530.409,Z 414.814,A -85,B 0,C 180,E1 -1944.375,E2 -1944.375} C_VEL
LIN {X 0,Y 523.467,Z 401.67,A -85,B 0,C 180,E1 -1946.386,E2 -1946.386} C_VEL
LIN {X 0,Y 514.948,Z 386.681,A -85,B 0,C 180,E1 -1948.904,E2 -1948.904} C_VEL
LIN {X 0,Y 512.194,Z 381.833,A -85,B 0,C 180,E1 -1949.759,E2 -1949.759} C_VEL
LIN {X 0,Y 509.83,Z 377.513,A -85,B 0,C 180,E1 -1950.512,E2 -1950.512} C_VEL
LIN {X 0,Y 507.636,Z 373.588,A -85,B 0,C 180,E1 -1951.221,E2 -1951.221} C_VEL
LIN {X 0,Y 505.089,Z 369.517,A -85,B 0,C 180,E1 -1952.021,E2 -1952.021} C_VEL
LIN {X 0,Y 504.7,Z 367.869,A -85,B 0,C 180,E1 -1952.254,E2 -1952.254} C_VEL
LIN {X 0,Y 504.706,Z 367.865,A -85,B 0,C 180,E1 -1955.79,E2 -1955.79} C_VEL
LIN {X 0,Y 504.661,Z 367.87,A -85,B 0,C 180,E1 -1959.35,E2 -1959.35} C_VEL
LIN {X 0,Y 504.687,Z 367.866,A -85,B 0,C 180,E1 -1962.95,E2 -1962.95} C_VEL
LIN {X 0,Y 504.695,Z 367.866,A -85,B 0,C 180,E1 -1966.364,E2 -1966.364} C_VEL
LIN {X 0,Y 504.695,Z 367.869,A -85,B 0,C 180,E1 -1969.96,E2 -1969.96} C_VEL
LIN {X 0,Y 504.702,Z 367.87,A -85,B 0,C 180,E1 -1973.402,E2 -1973.402} C_VEL
LIN {X 0,Y 504.698,Z 367.87,A -85,B 0,C 180,E1 -1977.048,E2 -1977.048} C_VEL
LIN {X 0,Y 504.686,Z 367.869,A -85,B 0,C 180,E1 -1980.454,E2 -1980.454} C_VEL
LIN {X 0,Y 504.665,Z 367.874,A -85,B 0,C 180,E1 -1984.09,E2 -1984.09} C_VEL
LIN {X 0,Y 504.708,Z 367.869,A -85,B 0,C 180,E1 -1987.628,E2 -1987.628} C_VEL
LIN {X 0,Y 504.702,Z 367.871,A -85,B 0,C 180,E1 -1991.195,E2 -1991.195} C_VEL
LIN {X 0,Y 504.697,Z 367.868,A -85,B 0,C 180,E1 -1994.69,E2 -1994.69} C_VEL
LIN {X 0,Y 504.664,Z 367.869,A -85,B 0,C 180,E1 -1998.243,E2 -1998.243} C_VEL
LIN {X 0,Y 504.711,Z 367.864,A -85,B 0,C 180,E1 -2001.703,E2 -2001.703} C_VEL
LIN {X 0,Y 504.661,Z 367.871,A -85,B 0,C 180,E1 -2005.119,E2 -2005.119} C_VEL
LIN {X 0,Y 504.693,Z 367.866,A -85,B 0,C 180,E1 -2008.649,E2 -2008.649} C_VEL
LIN {X 0,Y 504.705,Z 367.864,A -85,B 0,C 180,E1 -2012.069,E2 -2012.069} C_VEL
LIN {X 0,Y 504.704,Z 367.85,A -85,B 0,C 180,E1 -2015.623,E2 -2015.623} C_VEL
LIN {X 0,Y 504.681,Z 367.872,A -85,B 0,C 180,E1 -2019.051,E2 -2019.051} C_VEL
LIN {X 0,Y 504.7,Z 367.851,A -85,B 0,C 180,E1 -2022.527,E2 -2022.527} C_VEL
LIN {X 0,Y 504.682,Z 367.867,A -85,B 0,C 180,E1 -2025.986,E2 -2025.986} C_VEL
LIN {X 0,Y 504.674,Z 367.875,A -85,B 0,C 180,E1 -2029.621,E2 -2029.621} C_VEL
LIN {X 0,Y 504.687,Z 367.871,A -85,B 0,C 180,E1 -2029.879,E2 -2029.879} C_VEL
LIN {X 0,Y 503.707,Z 367.985,A -85,B 0,C 180,E1 -2030.461,E2 -2030.461} C_VEL
LIN {X 0,Y 497.299,Z 368.783,A -85,B 0,C 180,E1 -2032.041,E2 -2032.041} C_VEL
LIN {X 0,Y 496.76,Z 368.858,A -85,B 0,C 180,E1 -2032.469,E2 -2032.469} C_VEL
LIN {X 0,Y 496.753,Z 368.902,A -85,B 0,C 180,E1 -2033.622,E2 -2033.622} C_VEL
LIN {X 0,Y 499.236,Z 375.399,A -85,B 0,C 180,E1 -2034.305,E2 -2034.305} C_VEL
LIN {X 0,Y 507.393,Z 396.568,A -85,B 0,C 180,E1 -2036.569,E2 -2036.569} C_VEL
LIN {X 0,Y 506.481,Z 425.212,A -85,B 0,C 180,E1 -2038.788,E2 -2038.788} C_VEL
LIN {X 0,Y 505.188,Z 466.097,A -85,B 0,C 180,E1 -2041.834,E2 -2041.834} C_VEL
LIN {X 0,Y 505.073,Z 480.997,A -85,B 0,C 180,E1 -2042.842,E2 -2042.842} C_VEL
LIN {X 0,Y 506.183,Z 489.715,A -85,B 0,C 180,E1 -2043.047,E2 -2043.047} C_VEL
LIN {X 0,Y 504.008,Z 688.787,A -85,B 0,C 180,E1 -2046.058,E2 -2046.058} C_VEL
LIN {X 0,Y 503.651,Z 707.131,A -85,B 0,C 180,E1 -2046.539,E2 -2046.539} C_VEL
LIN {X 0,Y 503.097,Z 724.585,A -85,B 0,C 180,E1 -2047.199,E2 -2047.199} C_VEL
LIN {X 0,Y 502.331,Z 742.139,A -85,B 0,C 180,E1 -2048.081,E2 -2048.081} C_VEL
LIN {X 0,Y 501.457,Z 758.783,A -85,B 0,C 180,E1 -2049.149,E2 -2049.149} C_VEL
LIN {X 0,Y 500.555,Z 774.4,A -85,B 0,C 180,E1 -2050.392,E2 -2050.392} C_VEL
LIN {X 0,Y 499.602,Z 788.986,A -85,B 0,C 180,E1 -2051.808,E2 -2051.808} C_VEL
LIN {X 0,Y 498.685,Z 802.603,A -85,B 0,C 180,E1 -2053.414,E2 -2053.414} C_VEL
LIN {X 0,Y 497.885,Z 814.482,A -85,B 0,C 180,E1 -2055.105,E2 -2055.105} C_VEL
LIN {X 0,Y 497.207,Z 825.335,A -85,B 0,C 180,E1 -2056.984,E2 -2056.984} C_VEL
LIN {X 0,Y 496.702,Z 834.658,A -85,B 0,C 180,E1 -2058.975,E2 -2058.975} C_VEL
LIN {X 0,Y 496.332,Z 842.446,A -85,B 0,C 180,E1 -2061.077,E2 -2061.077} C_VEL
LIN {X 0,Y 496.13,Z 848.645,A -85,B 0,C 180,E1 -2063.288,E2 -2063.288} C_VEL
LIN {X 0,Y 496.044,Z 852.972,A -85,B 0,C 180,E1 -2065.492,E2 -2065.492} C_VEL
LIN {X 0,Y 495.993,Z 855.569,A -85,B 0,C 180,E1 -2067.69,E2 -2067.69} C_VEL
LIN {X 0,Y 495.982,Z 856.511,A -85,B 0,C 180,E1 -2069.885,E2 -2069.885} C_VEL
LIN {X 0,Y 495.993,Z 855.753,A -85,B 0,C 180,E1 -2072.195,E2 -2072.195} C_VEL
LIN {X 0,Y 496.039,Z 853.314,A -85,B 0,C 180,E1 -2074.393,E2 -2074.393} C_VEL
LIN {X 0,Y 496.117,Z 849.141,A -85,B 0,C 180,E1 -2076.597,E2 -2076.597} C_VEL
LIN {X 0,Y 496.3,Z 843.487,A -85,B 0,C 180,E1 -2078.691,E2 -2078.691} C_VEL
LIN {X 0,Y 496.632,Z 835.988,A -85,B 0,C 180,E1 -2080.792,E2 -2080.792} C_VEL
LIN {X 0,Y 497.111,Z 826.978,A -85,B 0,C 180,E1 -2082.783,E2 -2082.783} C_VEL
LIN {X 0,Y 497.748,Z 816.478,A -85,B 0,C 180,E1 -2084.662,E2 -2084.662} C_VEL
LIN {X 0,Y 498.554,Z 804.462,A -85,B 0,C 180,E1 -2086.426,E2 -2086.426} C_VEL
LIN {X 0,Y 499.426,Z 791.367,A -85,B 0,C 180,E1 -2088.017,E2 -2088.017} C_VEL
LIN {X 0,Y 500.322,Z 777.74,A -85,B 0,C 180,E1 -2089.393,E2 -2089.393} C_VEL
LIN {X 0,Y 501.265,Z 762.176,A -85,B 0,C 180,E1 -2090.69,E2 -2090.69} C_VEL
LIN {X 0,Y 502.102,Z 746.687,A -85,B 0,C 180,E1 -2091.74,E2 -2091.74} C_VEL
LIN {X 0,Y 502.868,Z 730.32,A -85,B 0,C 180,E1 -2092.628,E2 -2092.628} C_VEL
LIN {X 0,Y 503.504,Z 712.281,A -85,B 0,C 180,E1 -2093.378,E2 -2093.378} C_VEL
LIN {X 0,Y 503.938,Z 694.06,A -85,B 0,C 180,E1 -2093.915,E2 -2093.915} C_VEL
LIN {X 0,Y 504.187,Z 672.531,A -85,B 0,C 180,E1 -2094.305,E2 -2094.305} C_VEL
LIN {X 0,Y 506.032,Z 486.902,A -85,B 0,C 180,E1 -2097.097,E2 -2097.097} C_VEL
LIN {X 0,Y 504.985,Z 480.15,A -85,B 0,C 180,E1 -2097.282,E2 -2097.282} C_VEL
LIN {X 0,Y 505.696,Z 446.496,A -85,B 0,C 180,E1 -2099.689,E2 -2099.689} C_VEL
LIN {X 0,Y 507.423,Z 401.572,A -85,B 0,C 180,E1 -2103.128,E2 -2103.128} C_VEL
LIN {X 0,Y 507.356,Z 396.594,A -85,B 0,C 180,E1 -2103.527,E2 -2103.527} C_VEL
LIN {X 0,Y 499.217,Z 375.386,A -85,B 0,C 180,E1 -2105.792,E2 -2105.792} C_VEL
LIN {X 0,Y 496.728,Z 368.864,A -85,B 0,C 180,E1 -2106.499,E2 -2106.499} C_VEL
LIN {X 0,Y 496.716,Z 368.857,A -85,B 0,C 180,E1 -2109.951,E2 -2109.951} C_VEL
LIN {X 0,Y 496.769,Z 368.849,A -85,B 0,C 180,E1 -2113.342,E2 -2113.342} C_VEL
LIN {X 0,Y 496.726,Z 368.861,A -85,B 0,C 180,E1 -2116.812,E2 -2116.812} C_VEL
LIN {X 0,Y 496.712,Z 368.856,A -85,B 0,C 180,E1 -2120.349,E2 -2120.349} C_VEL
LIN {X 0,Y 496.727,Z 368.978,A -85,B 0,C 180,E1 -2120.5,E2 -2120.5} C_VEL
LIN {X 0,Y 498.128,Z 372.476,A -85,B 0,C 180,E1 -2120.969,E2 -2120.969} C_VEL
LIN {X 0,Y 506.679,Z 393.357,A -85,B 0,C 180,E1 -2123.7,E2 -2123.7} C_VEL
LIN {X 0,Y 509.789,Z 401.932,A -85,B 0,C 180,E1 -2124.737,E2 -2124.737} C_VEL
LIN {X 0,Y 507.834,Z 441.506,A -85,B 0,C 180,E1 -2128.059,E2 -2128.059} C_VEL
LIN {X 0,Y 505.739,Z 483.601,A -85,B 0,C 180,E1 -2131.545,E2 -2131.545} C_VEL
LIN {X 0,Y 503.791,Z 527.54,A -85,B 0,C 180,E1 -2135.118,E2 -2135.118} C_VEL
LIN {X 0,Y 501.962,Z 573.183,A -85,B 0,C 180,E1 -2138.783,E2 -2138.783} C_VEL
LIN {X 0,Y 501.329,Z 594.118,A -85,B 0,C 180,E1 -2140.415,E2 -2140.415} C_VEL
LIN {X 0,Y 501.989,Z 601.89,A -85,B 0,C 180,E1 -2140.581,E2 -2140.581} C_VEL
LIN {X 0,Y 500.21,Z 738.1,A -85,B 0,C 180,E1 -2142.819,E2 -2142.819} C_VEL
LIN {X 0,Y 499.934,Z 754.931,A -85,B 0,C 180,E1 -2143.321,E2 -2143.321} C_VEL
LIN {X 0,Y 499.564,Z 769.602,A -85,B 0,C 180,E1 -2143.966,E2 -2143.966} C_VEL
LIN {X 0,Y 499.06,Z 784.482,A -85,B 0,C 180,E1 -2144.843,E2 -2144.843} C_VEL
LIN {X 0,Y 498.524,Z 798.365,A -85,B 0,C 180,E1 -2145.896,E2 -2145.896} C_VEL
LIN {X 0,Y 497.957,Z 811.663,A -85,B 0,C 180,E1 -2147.18,E2 -2147.18} C_VEL
LIN {X 0,Y 497.476,Z 822.84,A -85,B 0,C 180,E1 -2148.523,E2 -2148.523} C_VEL
LIN {X 0,Y 497.053,Z 832.906,A -85,B 0,C 180,E1 -2150.038,E2 -2150.038} C_VEL
LIN {X 0,Y 496.728,Z 841.544,A -85,B 0,C 180,E1 -2151.667,E2 -2151.667} C_VEL
LIN {X 0,Y 496.495,Z 848.611,A -85,B 0,C 180,E1 -2153.408,E2 -2153.408} C_VEL
LIN {X 0,Y 496.352,Z 854.157,A -85,B 0,C 180,E1 -2155.262,E2 -2155.262} C_VEL
LIN {X 0,Y 496.292,Z 857.794,A -85,B 0,C 180,E1 -2157.113,E2 -2157.113} C_VEL
LIN {X 0,Y 496.281,Z 859.792,A -85,B 0,C 180,E1 -2159.076,E2 -2159.076} C_VEL
LIN {X 0,Y 496.298,Z 859.974,A -85,B 0,C 180,E1 -2160.923,E2 -2160.923} C_VEL
LIN {X 0,Y 496.36,Z 858.339,A -85,B 0,C 180,E1 -2162.886,E2 -2162.886} C_VEL
LIN {X 0,Y 496.458,Z 855.081,A -85,B 0,C 180,E1 -2164.736,E2 -2164.736} C_VEL
LIN {X 0,Y 496.681,Z 849.58,A -85,B 0,C 180,E1 -2166.705,E2 -2166.705} C_VEL
LIN {X 0,Y 496.976,Z 842.773,A -85,B 0,C 180,E1 -2168.445,E2 -2168.445} C_VEL
LIN {X 0,Y 497.364,Z 834.501,A -85,B 0,C 180,E1 -2170.072,E2 -2170.072} C_VEL
LIN {X 0,Y 497.841,Z 824.747,A -85,B 0,C 180,E1 -2171.586,E2 -2171.586} C_VEL
LIN {X 0,Y 498.427,Z 812.922,A -85,B 0,C 180,E1 -2173.042,E2 -2173.042} C_VEL
LIN {X 0,Y 499.012,Z 800.371,A -85,B 0,C 180,E1 -2174.267,E2 -2174.267} C_VEL
LIN {X 0,Y 499.565,Z 786.779,A -85,B 0,C 180,E1 -2175.319,E2 -2175.319} C_VEL
LIN {X 0,Y 500.009,Z 773.215,A -85,B 0,C 180,E1 -2176.138,E2 -2176.138} C_VEL
LIN {X 0,Y 500.367,Z 757.389,A -85,B 0,C 180,E1 -2176.842,E2 -2176.842} C_VEL
LIN {X 0,Y 500.569,Z 741.778,A -85,B 0,C 180,E1 -2177.318,E2 -2177.318} C_VEL
LIN {X 0,Y 502.582,Z 653.938,A -85,B 0,C 180,E1 -2179.02,E2 -2179.02} C_VEL
LIN {X 0,Y 504.481,Z 604.582,A -85,B 0,C 180,E1 -2180.052,E2 -2180.052} C_VEL
LIN {X 0,Y 505.535,Z 600.152,A -85,B 0,C 180,E1 -2180.365,E2 -2180.365} C_VEL
LIN {X 0,Y 509.143,Z 559.156,A -85,B 0,C 180,E1 -2183.985,E2 -2183.985} C_VEL
LIN {X 0,Y 513.986,Z 518.735,A -85,B 0,C 180,E1 -2187.734,E2 -2187.734} C_VEL
LIN {X 0,Y 518.857,Z 489.765,A -85,B 0,C 180,E1 -2190.579,E2 -2190.579} C_VEL
LIN {X 0,Y 524.523,Z 465.716,A -85,B 0,C 180,E1 -2193.102,E2 -2193.102} C_VEL
LIN {X 0,Y 530.803,Z 447.328,A -85,B 0,C 180,E1 -2195.198,E2 -2195.198} C_VEL
LIN {X 0,Y 534.263,Z 439.829,A -85,B 0,C 180,E1 -2196.122,E2 -2196.122} C_VEL
LIN {X 0,Y 526.91,Z 451.565,A -85,B 0,C 180,E1 -2197.336,E2 -2197.336} C_VEL
LIN {X 0,Y 521.792,Z 463.496,A -85,B 0,C 180,E1 -2198.573,E2 -2198.573} C_VEL
LIN {X 0,Y 519.013,Z 474.978,A -85,B 0,C 180,E1 -2199.766,E2 -2199.766} C_VEL
LIN {X 0,Y 518.297,Z 486.536,A -85,B 0,C 180,E1 -2200.988,E2 -2200.988} C_VEL
LIN {X 0,Y 519.643,Z 497.808,A -85,B 0,C 180,E1 -2202.201,E2 -2202.201} C_VEL
LIN {X 0,Y 522.91,Z 508.126,A -85,B 0,C 180,E1 -2203.349,E2 -2203.349} C_VEL
LIN {X 0,Y 528.107,Z 517.8,A -85,B 0,C 180,E1 -2204.468,E2 -2204.468} C_VEL
LIN {X 0,Y 535.169,Z 526.615,A -85,B 0,C 180,E1 -2205.536,E2 -2205.536} C_VEL
LIN {X 0,Y 544.058,Z 534.5,A -85,B 0,C 180,E1 -2206.545,E2 -2206.545} C_VEL
LIN {X 0,Y 553.916,Z 540.85,A -85,B 0,C 180,E1 -2207.431,E2 -2207.431} C_VEL
LIN {X 0,Y 564.747,Z 545.76,A -85,B 0,C 180,E1 -2208.264,E2 -2208.264} C_VEL
LIN {X 0,Y 569.319,Z 546.916,A -85,B 0,C 180,E1 -2208.735,E2 -2208.735} C_VEL
LIN {X 0,Y 572.738,Z 547.028,A -85,B 0,C 180,E1 -2209.258,E2 -2209.258} C_VEL
LIN {X 0,Y 575.221,Z 546.099,A -85,B 0,C 180,E1 -2209.89,E2 -2209.89} C_VEL
LIN {X 0,Y 576.143,Z 544.302,A -85,B 0,C 180,E1 -2210.503,E2 -2210.503} C_VEL
LIN {X 0,Y 575.543,Z 541.546,A -85,B 0,C 180,E1 -2211.125,E2 -2211.125} C_VEL
LIN {X 0,Y 568.61,Z 569.316,A -85,B 0,C 180,E1 -2211.49,E2 -2211.49} C_VEL
LIN {X 0,Y 564.616,Z 583.071,A -85,B 0,C 180,E1 -2211.811,E2 -2211.811} C_VEL
LIN {X 0,Y 563.59,Z 586.51,A -85,B 0,C 180,E1 -2211.864,E2 -2211.864} C_VEL
LIN {X 0,Y 556.045,Z 607.983,A -85,B 0,C 180,E1 -2211.961,E2 -2211.961} C_VEL
LIN {X 0,Y 546.602,Z 629.71,A -85,B 0,C 180,E1 -2212.165,E2 -2212.165} C_VEL
LIN {X 0,Y 538.072,Z 648.042,A -85,B 0,C 180,E1 -2212.51,E2 -2212.51} C_VEL
LIN {X 0,Y 531.841,Z 662.974,A -85,B 0,C 180,E1 -2212.948,E2 -2212.948} C_VEL
LIN {X 0,Y 528.697,Z 672.388,A -85,B 0,C 180,E1 -2213.301,E2 -2213.301} C_VEL
LIN {X 0,Y 522.443,Z 686.513,A -85,B 0,C 180,E1 -2213.745,E2 -2213.745} C_VEL
LIN {X 0,Y 518.491,Z 698.925,A -85,B 0,C 180,E1 -2214.246,E2 -2214.246} C_VEL
LIN {X 0,Y 514.276,Z 712.353,A -85,B 0,C 180,E1 -2214.798,E2 -2214.798} C_VEL
LIN {X 0,Y 512.177,Z 721.74,A -85,B 0,C 180,E1 -2215.196,E2 -2215.196} C_VEL
LIN {X 0,Y 511.638,Z 762.179,A -85,B 0,C 180,E1 -2215.825,E2 -2215.825} C_VEL
LIN {X 0,Y 510.845,Z 783.222,A -85,B 0,C 180,E1 -2216.343,E2 -2216.343} C_VEL
LIN {X 0,Y 509.738,Z 804.792,A -85,B 0,C 180,E1 -2217.09,E2 -2217.09} C_VEL
LIN {X 0,Y 508.489,Z 825.075,A -85,B 0,C 180,E1 -2217.999,E2 -2217.999} C_VEL
LIN {X 0,Y 506.965,Z 845.809,A -85,B 0,C 180,E1 -2219.15,E2 -2219.15} C_VEL
LIN {X 0,Y 505.403,Z 865.909,A -85,B 0,C 180,E1 -2220.513,E2 -2220.513} C_VEL
LIN {X 0,Y 503.752,Z 885.095,A -85,B 0,C 180,E1 -2222.068,E2 -2222.068} C_VEL
LIN {X 0,Y 502.156,Z 903.5,A -85,B 0,C 180,E1 -2223.83,E2 -2223.83} C_VEL
LIN {X 0,Y 500.713,Z 920.231,A -85,B 0,C 180,E1 -2225.71,E2 -2225.71} C_VEL
LIN {X 0,Y 499.411,Z 935.908,A -85,B 0,C 180,E1 -2227.765,E2 -2227.765} C_VEL
LIN {X 0,Y 498.325,Z 950.062,A -85,B 0,C 180,E1 -2229.934,E2 -2229.934} C_VEL
LIN {X 0,Y 497.472,Z 962.743,A -85,B 0,C 180,E1 -2232.211,E2 -2232.211} C_VEL
LIN {X 0,Y 496.799,Z 974.401,A -85,B 0,C 180,E1 -2234.713,E2 -2234.713} C_VEL
LIN {X 0,Y 496.367,Z 983.927,A -85,B 0,C 180,E1 -2237.198,E2 -2237.198} C_VEL
LIN {X 0,Y 496.1,Z 991.893,A -85,B 0,C 180,E1 -2239.784,E2 -2239.784} C_VEL
LIN {X 0,Y 495.967,Z 997.678,A -85,B 0,C 180,E1 -2242.237,E2 -2242.237} C_VEL
LIN {X 0,Y 495.91,Z 1001.818,A -85,B 0,C 180,E1 -2244.678,E2 -2244.678} C_VEL
LIN {X 0,Y 495.895,Z 1004.363,A -85,B 0,C 180,E1 -2247.11,E2 -2247.11} C_VEL
LIN {X 0,Y 495.894,Z 1005.369,A -85,B 0,C 180,E1 -2249.307,E2 -2249.307} C_VEL
LIN {X 0,Y 495.901,Z 1005.109,A -85,B 0,C 180,E1 -2251.733,E2 -2251.733} C_VEL
LIN {X 0,Y 495.92,Z 1003.122,A -85,B 0,C 180,E1 -2254.278,E2 -2254.278} C_VEL
LIN {X 0,Y 495.952,Z 999.639,A -85,B 0,C 180,E1 -2256.715,E2 -2256.715} C_VEL
LIN {X 0,Y 496.039,Z 994.594,A -85,B 0,C 180,E1 -2259.162,E2 -2259.162} C_VEL
LIN {X 0,Y 496.229,Z 987.427,A -85,B 0,C 180,E1 -2261.742,E2 -2261.742} C_VEL
LIN {X 0,Y 496.574,Z 978.721,A -85,B 0,C 180,E1 -2264.22,E2 -2264.22} C_VEL
LIN {X 0,Y 497.101,Z 968.565,A -85,B 0,C 180,E1 -2266.595,E2 -2266.595} C_VEL
LIN {X 0,Y 497.86,Z 956.639,A -85,B 0,C 180,E1 -2268.931,E2 -2268.931} C_VEL
LIN {X 0,Y 498.834,Z 943.292,A -85,B 0,C 180,E1 -2271.148,E2 -2271.148} C_VEL
LIN {X 0,Y 500.066,Z 927.941,A -85,B 0,C 180,E1 -2273.321,E2 -2273.321} C_VEL
LIN {X 0,Y 501.524,Z 910.855,A -85,B 0,C 180,E1 -2275.381,E2 -2275.381} C_VEL
LIN {X 0,Y 503.124,Z 892.469,A -85,B 0,C 180,E1 -2277.262,E2 -2277.262} C_VEL
LIN {X 0,Y 504.75,Z 873.513,A -85,B 0,C 180,E1 -2278.903,E2 -2278.903} C_VEL
LIN {X 0,Y 506.321,Z 854.329,A -85,B 0,C 180,E1 -2280.301,E2 -2280.301} C_VEL
LIN {X 0,Y 507.822,Z 834.406,A -85,B 0,C 180,E1 -2281.512,E2 -2281.512} C_VEL
LIN {X 0,Y 509.228,Z 813.477,A -85,B 0,C 180,E1 -2282.547,E2 -2282.547} C_VEL
LIN {X 0,Y 510.446,Z 791.809,A -85,B 0,C 180,E1 -2283.387,E2 -2283.387} C_VEL
LIN {X 0,Y 511.385,Z 770.024,A -85,B 0,C 180,E1 -2284.01,E2 -2284.01} C_VEL
LIN {X 0,Y 511.957,Z 746.359,A -85,B 0,C 180,E1 -2284.444,E2 -2284.444} C_VEL
LIN {X 0,Y 512.317,Z 720.574,A -85,B 0,C 180,E1 -2284.844,E2 -2284.844} C_VEL
LIN {X 0,Y 516.703,Z 704.266,A -85,B 0,C 180,E1 -2285.555,E2 -2285.555} C_VEL
LIN {X 0,Y 519.624,Z 694.889,A -85,B 0,C 180,E1 -2285.936,E2 -2285.936} C_VEL
LIN {X 0,Y 524.487,Z 681.512,A -85,B 0,C 180,E1 -2286.429,E2 -2286.429} C_VEL
LIN {X 0,Y 529.148,Z 671.369,A -85,B 0,C 180,E1 -2286.73,E2 -2286.73} C_VEL
LIN {X 0,Y 533.385,Z 658.952,A -85,B 0,C 180,E1 -2287.186,E2 -2287.186} C_VEL
LIN {X 0,Y 540.914,Z 641.869,A -85,B 0,C 180,E1 -2287.629,E2 -2287.629} C_VEL
LIN {X 0,Y 550.329,Z 621.544,A -85,B 0,C 180,E1 -2287.93,E2 -2287.93} C_VEL
LIN {X 0,Y 559.213,Z 599.619,A -85,B 0,C 180,E1 -2288.086,E2 -2288.086} C_VEL
LIN {X 0,Y 564.445,Z 583.652,A -85,B 0,C 180,E1 -2288.17,E2 -2288.17} C_VEL
LIN {X 0,Y 568.347,Z 570.246,A -85,B 0,C 180,E1 -2288.494,E2 -2288.494} C_VEL
LIN {X 0,Y 574.28,Z 547.057,A -85,B 0,C 180,E1 -2288.797,E2 -2288.797} C_VEL
LIN {X 0,Y 575.542,Z 541.545,A -85,B 0,C 180,E1 -2288.875,E2 -2288.875} C_VEL
LIN {X 0,Y 576.143,Z 544.3,A -85,B 0,C 180,E1 -2289.497,E2 -2289.497} C_VEL
LIN {X 0,Y 575.221,Z 546.1,A -85,B 0,C 180,E1 -2290.11,E2 -2290.11} C_VEL
LIN {X 0,Y 572.737,Z 547.029,A -85,B 0,C 180,E1 -2290.742,E2 -2290.742} C_VEL
LIN {X 0,Y 569.319,Z 546.916,A -85,B 0,C 180,E1 -2291.265,E2 -2291.265} C_VEL
LIN {X 0,Y 562.995,Z 545.202,A -85,B 0,C 180,E1 -2291.916,E2 -2291.916} C_VEL
LIN {X 0,Y 553.301,Z 540.915,A -85,B 0,C 180,E1 -2292.957,E2 -2292.957} C_VEL
LIN {X 0,Y 544.388,Z 534.893,A -85,B 0,C 180,E1 -2294.1,E2 -2294.1} C_VEL
LIN {X 0,Y 536.942,Z 527.487,A -85,B 0,C 180,E1 -2295.261,E2 -2295.261} C_VEL
LIN {X 0,Y 530.938,Z 518.768,A -85,B 0,C 180,E1 -2296.43,E2 -2296.43} C_VEL
LIN {X 0,Y 526.066,Z 507.974,A -85,B 0,C 180,E1 -2297.675,E2 -2297.675} C_VEL
LIN {X 0,Y 522.953,Z 496.098,A -85,B 0,C 180,E1 -2298.877,E2 -2298.877} C_VEL
LIN {X 0,Y 521.204,Z 480.803,A -85,B 0,C 180,E1 -2300.233,E2 -2300.233} C_VEL
LIN {X 0,Y 521.273,Z 463.526,A -85,B 0,C 180,E1 -2301.577,E2 -2301.577} C_VEL
